LIN {X 0,Y 417.271,Z 465.296,A -85,B 0,C 180,E1 -10175.316,E2 -10175.316} C_VEL
LIN {X 0,Y 417.317,Z 461.12,A -85,B 0,C 180,E1 -10176.771,E2 -10176.771} C_VEL
LIN {X 0,Y 417.422,Z 454.683,A -85,B 0,C 180,E1 -10178.472,E2 -10178.472} C_VEL
LIN {X 0,Y 417.63,Z 447.667,A -85,B 0,C 180,E1 -10179.933,E2 -10179.933} C_VEL
LIN {X 0,Y 418.109,Z 438.94,A -85,B 0,C 180,E1 -10181.392,E2 -10181.392} C_VEL
LIN {X 0,Y 418.694,Z 429.948,A -85,B 0,C 180,E1 -10182.605,E2 -10182.605} C_VEL
LIN {X 0,Y 419.338,Z 418.893,A -85,B 0,C 180,E1 -10183.818,E2 -10183.818} C_VEL
LIN {X 0,Y 420.032,Z 407.756,A -85,B 0,C 180,E1 -10184.784,E2 -10184.784} C_VEL
LIN {X 0,Y 420.914,Z 395.292,A -85,B 0,C 180,E1 -10185.62,E2 -10185.62} C_VEL
LIN {X 0,Y 421.545,Z 382.66,A -85,B 0,C 180,E1 -10186.247,E2 -10186.247} C_VEL
LIN {X 0,Y 422.133,Z 369.345,A -85,B 0,C 180,E1 -10186.69,E2 -10186.69} C_VEL
LIN {X 0,Y 423.204,Z 286.093,A -85,B 0,C 180,E1 -10188.305,E2 -10188.305} C_VEL
LIN {X 0,Y 420.595,Z 264.034,A -85,B 0,C 180,E1 -10188.899,E2 -10188.899} C_VEL
LIN {X 0,Y 420.271,Z 261.318,A -85,B 0,C 180,E1 -10189.016,E2 -10189.016} C_VEL
LIN {X 0,Y 421.665,Z 236.885,A -85,B 0,C 180,E1 -10192.542,E2 -10192.542} C_VEL
LIN {X 0,Y 423.214,Z 213.553,A -85,B 0,C 180,E1 -10195.973,E2 -10195.973} C_VEL
LIN {X 0,Y 420.894,Z 202.341,A -85,B 0,C 180,E1 -10197.875,E2 -10197.875} C_VEL
LIN {X 0,Y 418.276,Z 192.511,A -85,B 0,C 180,E1 -10199.696,E2 -10199.696} C_VEL
LIN {X 0,Y 418.261,Z 192.387,A -85,B 0,C 180,E1 -10202.844,E2 -10202.844} C_VEL
LIN {X 0,Y 418.247,Z 192.387,A -85,B 0,C 180,E1 -10206.238,E2 -10206.238} C_VEL
LIN {X 0,Y 418.203,Z 192.393,A -85,B 0,C 180,E1 -10209.688,E2 -10209.688} C_VEL
LIN {X 0,Y 418.215,Z 192.39,A -85,B 0,C 180,E1 -10212.318,E2 -10212.318} C_VEL
LIN {X 0,Y 418.239,Z 192.391,A -85,B 0,C 180,E1 -10215.109,E2 -10215.109} C_VEL
LIN {X 0,Y 418.237,Z 192.384,A -85,B 0,C 180,E1 -10217.766,E2 -10217.766} C_VEL
LIN {X 0,Y 418.248,Z 192.385,A -85,B 0,C 180,E1 -10220.621,E2 -10220.621} C_VEL
LIN {X 0,Y 418.245,Z 192.384,A -85,B 0,C 180,E1 -10223.976,E2 -10223.976} C_VEL
LIN {X 0,Y 418.26,Z 192.386,A -85,B 0,C 180,E1 -10227.156,E2 -10227.156} C_VEL
LIN {X 0,Y 418.271,Z 192.383,A -85,B 0,C 180,E1 -10230.895,E2 -10230.895} C_VEL
LIN {X 0,Y 418.271,Z 192.383,A -85,B 0,C 180,E1 -10234.095,E2 -10234.095} C_VEL
LIN {X 0,Y 418.24,Z 192.386,A -85,B 0,C 180,E1 -10237.263,E2 -10237.263} C_VEL
LIN {X 0,Y 418.285,Z 192.385,A -85,B 0,C 180,E1 -10240.364,E2 -10240.364} C_VEL
LIN {X 0,Y 418.318,Z 192.377,A -85,B 0,C 180,E1 -10243.404,E2 -10243.404} C_VEL
LIN {X 0,Y 418.348,Z 192.373,A -85,B 0,C 180,E1 -10246.999,E2 -10246.999} C_VEL
LIN {X 0,Y 418.341,Z 192.377,A -85,B 0,C 180,E1 -10250.328,E2 -10250.328} C_VEL
LIN {X 0,Y 418.46,Z 192.36,A -85,B 0,C 180,E1 -10253.248,E2 -10253.248} C_VEL
LIN {X 0,Y 418.334,Z 192.378,A -85,B 0,C 180,E1 -10255.181,E2 -10255.181} C_VEL
LIN {X 0,Y 418.456,Z 192.55,A -85,B 0,C 180,E1 -10256.871,E2 -10256.871} C_VEL
LIN {X 0,Y 420.63,Z 201.709,A -85,B 0,C 180,E1 -10258.803,E2 -10258.803} C_VEL
LIN {X 0,Y 420.547,Z 211.888,A -85,B 0,C 180,E1 -10260.718,E2 -10260.718} C_VEL
LIN {X 0,Y 420.179,Z 229.574,A -85,B 0,C 180,E1 -10264.016,E2 -10264.016} C_VEL
LIN {X 0,Y 423.338,Z 244.848,A -85,B 0,C 180,E1 -10264.582,E2 -10264.582} C_VEL
LIN {X 0,Y 421.949,Z 313.811,A -85,B 0,C 180,E1 -10266.125,E2 -10266.125} C_VEL
LIN {X 0,Y 421.711,Z 325.601,A -85,B 0,C 180,E1 -10266.579,E2 -10266.579} C_VEL
LIN {X 0,Y 421.311,Z 336.524,A -85,B 0,C 180,E1 -10267.187,E2 -10267.187} C_VEL
LIN {X 0,Y 420.865,Z 346.473,A -85,B 0,C 180,E1 -10267.918,E2 -10267.918} C_VEL
LIN {X 0,Y 420.345,Z 356.216,A -85,B 0,C 180,E1 -10268.841,E2 -10268.841} C_VEL
LIN {X 0,Y 419.827,Z 364.922,A -85,B 0,C 180,E1 -10269.88,E2 -10269.88} C_VEL
LIN {X 0,Y 419.243,Z 373.147,A -85,B 0,C 180,E1 -10271.115,E2 -10271.115} C_VEL
LIN {X 0,Y 418.796,Z 379.629,A -85,B 0,C 180,E1 -10272.354,E2 -10272.354} C_VEL
LIN {X 0,Y 418.393,Z 384.792,A -85,B 0,C 180,E1 -10273.601,E2 -10273.601} C_VEL
LIN {X 0,Y 418.019,Z 389.504,A -85,B 0,C 180,E1 -10275.105,E2 -10275.105} C_VEL
LIN {X 0,Y 417.796,Z 392.747,A -85,B 0,C 180,E1 -10276.616,E2 -10276.616} C_VEL
LIN {X 0,Y 417.651,Z 394.16,A -85,B 0,C 180,E1 -10277.631,E2 -10277.631} C_VEL
LIN {X 0,Y 417.524,Z 395.021,A -85,B 0,C 180,E1 -10278.651,E2 -10278.651} C_VEL
LIN {X 0,Y 417.469,Z 395.273,A -85,B 0,C 180,E1 -10279.675,E2 -10279.675} C_VEL
LIN {X 0,Y 417.425,Z 394.957,A -85,B 0,C 180,E1 -10280.705,E2 -10280.705} C_VEL
LIN {X 0,Y 417.497,Z 393.456,A -85,B 0,C 180,E1 -10282.203,E2 -10282.203} C_VEL
LIN {X 0,Y 417.655,Z 390.389,A -85,B 0,C 180,E1 -10283.819,E2 -10283.819} C_VEL
LIN {X 0,Y 417.803,Z 387.549,A -85,B 0,C 180,E1 -10284.868,E2 -10284.868} C_VEL
LIN {X 0,Y 418.077,Z 381.826,A -85,B 0,C 180,E1 -10286.453,E2 -10286.453} C_VEL
LIN {X 0,Y 418.354,Z 375.584,A -85,B 0,C 180,E1 -10287.759,E2 -10287.759} C_VEL
LIN {X 0,Y 418.706,Z 369.068,A -85,B 0,C 180,E1 -10288.853,E2 -10288.853} C_VEL
LIN {X 0,Y 419.139,Z 360.148,A -85,B 0,C 180,E1 -10290.05,E2 -10290.05} C_VEL
LIN {X 0,Y 419.518,Z 351.23,A -85,B 0,C 180,E1 -10291.006,E2 -10291.006} C_VEL
LIN {X 0,Y 419.96,Z 340.418,A -85,B 0,C 180,E1 -10291.911,E2 -10291.911} C_VEL
LIN {X 0,Y 420.333,Z 328.992,A -85,B 0,C 180,E1 -10292.63,E2 -10292.63} C_VEL
LIN {X 0,Y 420.541,Z 317.102,A -85,B 0,C 180,E1 -10293.164,E2 -10293.164} C_VEL
LIN {X 0,Y 420.702,Z 305.658,A -85,B 0,C 180,E1 -10293.49,E2 -10293.49} C_VEL
LIN {X 0,Y 421.451,Z 242.868,A -85,B 0,C 180,E1 -10294.748,E2 -10294.748} C_VEL
LIN {X 0,Y 419.042,Z 228.513,A -85,B 0,C 180,E1 -10295.14,E2 -10295.14} C_VEL
LIN {X 0,Y 419.063,Z 227.046,A -85,B 0,C 180,E1 -10295.35,E2 -10295.35} C_VEL
LIN {X 0,Y 419.499,Z 211.477,A -85,B 0,C 180,E1 -10298.613,E2 -10298.613} C_VEL
LIN {X 0,Y 419.772,Z 201.372,A -85,B 0,C 180,E1 -10300.764,E2 -10300.764} C_VEL
LIN {X 0,Y 418.633,Z 194.184,A -85,B 0,C 180,E1 -10302.381,E2 -10302.381} C_VEL
LIN {X 0,Y 418.268,Z 192.411,A -85,B 0,C 180,E1 -10302.87,E2 -10302.87} C_VEL
LIN {X 0,Y 418.208,Z 192.392,A -85,B 0,C 180,E1 -10306.27,E2 -10306.27} C_VEL
LIN {X 0,Y 418.221,Z 192.387,A -85,B 0,C 180,E1 -10309.13,E2 -10309.13} C_VEL
LIN {X 0,Y 418.225,Z 192.387,A -85,B 0,C 180,E1 -10312.166,E2 -10312.166} C_VEL
LIN {X 0,Y 418.264,Z 192.385,A -85,B 0,C 180,E1 -10315.419,E2 -10315.419} C_VEL
LIN {X 0,Y 418.209,Z 192.387,A -85,B 0,C 180,E1 -10318.603,E2 -10318.603} C_VEL
LIN {X 0,Y 418.291,Z 192.379,A -85,B 0,C 180,E1 -10321.936,E2 -10321.936} C_VEL
LIN {X 0,Y 418.288,Z 192.381,A -85,B 0,C 180,E1 -10325.162,E2 -10325.162} C_VEL
LIN {X 0,Y 418.232,Z 192.384,A -85,B 0,C 180,E1 -10328.303,E2 -10328.303} C_VEL
LIN {X 0,Y 418.282,Z 192.385,A -85,B 0,C 180,E1 -10331.383,E2 -10331.383} C_VEL
LIN {X 0,Y 418.291,Z 192.377,A -85,B 0,C 180,E1 -10334.036,E2 -10334.036} C_VEL
LIN {X 0,Y 417.64,Z 192.462,A -85,B 0,C 180,E1 -10334.84,E2 -10334.84} C_VEL
LIN {X 0,Y 414.816,Z 192.81,A -85,B 0,C 180,E1 -10336.148,E2 -10336.148} C_VEL
LIN {X 0,Y 412.412,Z 193.115,A -85,B 0,C 180,E1 -10337.203,E2 -10337.203} C_VEL
LIN {X 0,Y 411.367,Z 193.24,A -85,B 0,C 180,E1 -10338.019,E2 -10338.019} C_VEL
LIN {X 0,Y 411.276,Z 193.251,A -85,B 0,C 180,E1 -10338.295,E2 -10338.295} C_VEL
LIN {X 0,Y 411.48,Z 193.225,A -85,B 0,C 180,E1 -10342.146,E2 -10342.146} C_VEL
LIN {X 0,Y 411.474,Z 193.226,A -85,B 0,C 180,E1 -10344.117,E2 -10344.117} C_VEL
LIN {X 0,Y 411.511,Z 193.221,A -85,B 0,C 180,E1 -10348.042,E2 -10348.042} C_VEL
LIN {X 0,Y 411.64,Z 193.205,A -85,B 0,C 180,E1 -10349.999,E2 -10349.999} C_VEL
LIN {X 0,Y 411.463,Z 193.233,A -85,B 0,C 180,E1 -10352.936,E2 -10352.936} C_VEL
LIN {X 0,Y 411.448,Z 193.235,A -85,B 0,C 180,E1 -10356.866,E2 -10356.866} C_VEL
LIN {X 0,Y 411.29,Z 193.249,A -85,B 0,C 180,E1 -10359.838,E2 -10359.838} C_VEL
LIN {X 0,Y 411.301,Z 193.252,A -85,B 0,C 180,E1 -10363.103,E2 -10363.103} C_VEL
LIN {X 0,Y 411.253,Z 193.26,A -85,B 0,C 180,E1 -10366.888,E2 -10366.888} C_VEL
LIN {X 0,Y 411.225,Z 193.257,A -85,B 0,C 180,E1 -10369.986,E2 -10369.986} C_VEL
LIN {X 0,Y 411.198,Z 193.263,A -85,B 0,C 180,E1 -10373.147,E2 -10373.147} C_VEL
LIN {X 0,Y 411.233,Z 193.26,A -85,B 0,C 180,E1 -10376.38,E2 -10376.38} C_VEL
LIN {X 0,Y 411.194,Z 193.261,A -85,B 0,C 180,E1 -10379.712,E2 -10379.712} C_VEL
LIN {X 0,Y 411.2,Z 193.261,A -85,B 0,C 180,E1 -10383.155,E2 -10383.155} C_VEL
LIN {X 0,Y 411.189,Z 193.268,A -85,B 0,C 180,E1 -10386.553,E2 -10386.553} C_VEL
LIN {X 0,Y 411.22,Z 193.258,A -85,B 0,C 180,E1 -10389.73,E2 -10389.73} C_VEL
LIN {X 0,Y 411.214,Z 193.259,A -85,B 0,C 180,E1 -10393.127,E2 -10393.127} C_VEL
LIN {X 0,Y 411.165,Z 193.266,A -85,B 0,C 180,E1 -10395.88,E2 -10395.88} C_VEL
LIN {X 0,Y 411.203,Z 193.26,A -85,B 0,C 180,E1 -10399.499,E2 -10399.499} C_VEL
LIN {X 0,Y 411.195,Z 193.265,A -85,B 0,C 180,E1 -10402.027,E2 -10402.027} C_VEL
LIN {X 0,Y 411.198,Z 193.262,A -85,B 0,C 180,E1 -10405.666,E2 -10405.666} C_VEL
LIN {X 0,Y 411.193,Z 193.261,A -85,B 0,C 180,E1 -10409.153,E2 -10409.153} C_VEL
LIN {X 0,Y 411.251,Z 193.256,A -85,B 0,C 180,E1 -10412.522,E2 -10412.522} C_VEL
LIN {X 0,Y 411.218,Z 193.262,A -85,B 0,C 180,E1 -10415.785,E2 -10415.785} C_VEL
LIN {X 0,Y 411.188,Z 193.262,A -85,B 0,C 180,E1 -10418.966,E2 -10418.966} C_VEL
LIN {X 0,Y 411.245,Z 193.26,A -85,B 0,C 180,E1 -10422.085,E2 -10422.085} C_VEL
LIN {X 0,Y 411.256,Z 193.253,A -85,B 0,C 180,E1 -10425.148,E2 -10425.148} C_VEL
LIN {X 0,Y 411.276,Z 193.254,A -85,B 0,C 180,E1 -10428.168,E2 -10428.168} C_VEL
LIN {X 0,Y 411.432,Z 193.234,A -85,B 0,C 180,E1 -10432.189,E2 -10432.189} C_VEL
LIN {X 0,Y 411.466,Z 193.23,A -85,B 0,C 180,E1 -10434.118,E2 -10434.118} C_VEL
LIN {X 0,Y 411.502,Z 193.226,A -85,B 0,C 180,E1 -10438.043,E2 -10438.043} C_VEL
LIN {X 0,Y 411.633,Z 193.209,A -85,B 0,C 180,E1 -10440,E2 -10440} C_VEL
LIN {X 0,Y 411.45,Z 193.23,A -85,B 0,C 180,E1 -10442.938,E2 -10442.938} C_VEL
LIN {X 0,Y 411.45,Z 193.23,A -85,B 0,C 180,E1 -10446.868,E2 -10446.868} C_VEL
LIN {X 0,Y 411.346,Z 193.243,A -85,B 0,C 180,E1 -10448.846,E2 -10448.846} C_VEL
LIN {X 0,Y 411.276,Z 193.254,A -85,B 0,C 180,E1 -10451.833,E2 -10451.833} C_VEL
LIN {X 0,Y 411.252,Z 193.255,A -85,B 0,C 180,E1 -10454.853,E2 -10454.853} C_VEL
LIN {X 0,Y 411.245,Z 193.256,A -85,B 0,C 180,E1 -10457.916,E2 -10457.916} C_VEL
LIN {X 0,Y 411.19,Z 193.265,A -85,B 0,C 180,E1 -10461.035,E2 -10461.035} C_VEL
LIN {X 0,Y 411.22,Z 193.258,A -85,B 0,C 180,E1 -10464.216,E2 -10464.216} C_VEL
LIN {X 0,Y 411.253,Z 193.258,A -85,B 0,C 180,E1 -10467.479,E2 -10467.479} C_VEL
LIN {X 0,Y 411.183,Z 193.265,A -85,B 0,C 180,E1 -10470.849,E2 -10470.849} C_VEL
LIN {X 0,Y 411.199,Z 193.26,A -85,B 0,C 180,E1 -10474.335,E2 -10474.335} C_VEL
LIN {X 0,Y 411.188,Z 193.262,A -85,B 0,C 180,E1 -10477.975,E2 -10477.975} C_VEL
LIN {X 0,Y 411.159,Z 193.27,A -85,B 0,C 180,E1 -10481.229,E2 -10481.229} C_VEL
LIN {X 0,Y 411.172,Z 193.265,A -85,B 0,C 180,E1 -10484.491,E2 -10484.491} C_VEL
LIN {X 0,Y 411.17,Z 193.264,A -85,B 0,C 180,E1 -10488.195,E2 -10488.195} C_VEL
LIN {X 0,Y 411.208,Z 193.265,A -85,B 0,C 180,E1 -10490.776,E2 -10490.776} C_VEL
LIN {X 0,Y 411.195,Z 193.264,A -85,B 0,C 180,E1 -10494.472,E2 -10494.472} C_VEL
LIN {X 0,Y 411.206,Z 193.266,A -85,B 0,C 180,E1 -10496.874,E2 -10496.874} C_VEL
LIN {X 0,Y 411.263,Z 193.447,A -85,B 0,C 180,E1 -10500.405,E2 -10500.405} C_VEL
LIN {X 0,Y 415.049,Z 210.098,A -85,B 0,C 180,E1 -10503.317,E2 -10503.317} C_VEL
LIN {X 0,Y 415.807,Z 213.749,A -85,B 0,C 180,E1 -10503.932,E2 -10503.932} C_VEL
LIN {X 0,Y 414.983,Z 228.074,A -85,B 0,C 180,E1 -10506.139,E2 -10506.139} C_VEL
LIN {X 0,Y 413.235,Z 254.249,A -85,B 0,C 180,E1 -10510.115,E2 -10510.115} C_VEL
LIN {X 0,Y 412.767,Z 263.296,A -85,B 0,C 180,E1 -10511.448,E2 -10511.448} C_VEL
LIN {X 0,Y 415.274,Z 288.029,A -85,B 0,C 180,E1 -10512.03,E2 -10512.03} C_VEL
LIN {X 0,Y 414.314,Z 370.3,A -85,B 0,C 180,E1 -10513.589,E2 -10513.589} C_VEL
LIN {X 0,Y 413.823,Z 383.827,A -85,B 0,C 180,E1 -10514.044,E2 -10514.044} C_VEL
LIN {X 0,Y 413.289,Z 396.045,A -85,B 0,C 180,E1 -10514.655,E2 -10514.655} C_VEL
LIN {X 0,Y 412.62,Z 407.808,A -85,B 0,C 180,E1 -10515.45,E2 -10515.45} C_VEL
LIN {X 0,Y 412,Z 418.559,A -85,B 0,C 180,E1 -10516.378,E2 -10516.378} C_VEL
LIN {X 0,Y 411.554,Z 428.336,A -85,B 0,C 180,E1 -10517.425,E2 -10517.425} C_VEL
LIN {X 0,Y 411.037,Z 435.948,A -85,B 0,C 180,E1 -10518.411,E2 -10518.411} C_VEL
LIN {X 0,Y 410.635,Z 443.931,A -85,B 0,C 180,E1 -10519.648,E2 -10519.648} C_VEL
LIN {X 0,Y 410.332,Z 451.666,A -85,B 0,C 180,E1 -10521.133,E2 -10521.133} C_VEL
LIN {X 0,Y 410.256,Z 457.854,A -85,B 0,C 180,E1 -10522.619,E2 -10522.619} C_VEL
LIN {X 0,Y 410.195,Z 462.697,A -85,B 0,C 180,E1 -10524.1,E2 -10524.1} C_VEL
LIN {X 0,Y 410.153,Z 466.343,A -85,B 0,C 180,E1 -10525.578,E2 -10525.578} C_VEL
LIN {X 0,Y 410.337,Z 468.924,A -85,B 0,C 180,E1 -10527.055,E2 -10527.055} C_VEL
LIN {X 0,Y 410.289,Z 470.074,A -85,B 0,C 180,E1 -10528.037,E2 -10528.037} C_VEL
LIN {X 0,Y 410.211,Z 470.747,A -85,B 0,C 180,E1 -10529.019,E2 -10529.019} C_VEL
LIN {X 0,Y 410.211,Z 471.014,A -85,B 0,C 180,E1 -10530.001,E2 -10530.001} C_VEL
LIN {X 0,Y 410.212,Z 470.867,A -85,B 0,C 180,E1 -10530.982,E2 -10530.982} C_VEL
LIN {X 0,Y 410.287,Z 470.264,A -85,B 0,C 180,E1 -10531.964,E2 -10531.964} C_VEL
LIN {X 0,Y 410.293,Z 469.224,A -85,B 0,C 180,E1 -10532.946,E2 -10532.946} C_VEL
LIN {X 0,Y 410.208,Z 467.759,A -85,B 0,C 180,E1 -10533.93,E2 -10533.93} C_VEL
LIN {X 0,Y 410.177,Z 464.691,A -85,B 0,C 180,E1 -10535.408,E2 -10535.408} C_VEL
LIN {X 0,Y 410.25,Z 460.536,A -85,B 0,C 180,E1 -10536.888,E2 -10536.888} C_VEL
LIN {X 0,Y 410.332,Z 454.126,A -85,B 0,C 180,E1 -10538.62,E2 -10538.62} C_VEL
LIN {X 0,Y 410.577,Z 447.128,A -85,B 0,C 180,E1 -10540.106,E2 -10540.106} C_VEL
LIN {X 0,Y 411.103,Z 438.459,A -85,B 0,C 180,E1 -10541.589,E2 -10541.589} C_VEL
LIN {X 0,Y 411.731,Z 429.519,A -85,B 0,C 180,E1 -10542.821,E2 -10542.821} C_VEL
LIN {X 0,Y 412.344,Z 419.718,A -85,B 0,C 180,E1 -10543.931,E2 -10543.931} C_VEL
LIN {X 0,Y 413.035,Z 409.012,A -85,B 0,C 180,E1 -10544.914,E2 -10544.914} C_VEL
LIN {X 0,Y 413.956,Z 397.074,A -85,B 0,C 180,E1 -10545.763,E2 -10545.763} C_VEL
LIN {X 0,Y 414.627,Z 384.67,A -85,B 0,C 180,E1 -10546.431,E2 -10546.431} C_VEL
LIN {X 0,Y 415.25,Z 371.848,A -85,B 0,C 180,E1 -10546.912,E2 -10546.912} C_VEL
LIN {X 0,Y 415.607,Z 355.316,A -85,B 0,C 180,E1 -10547.277,E2 -10547.277} C_VEL
LIN {X 0,Y 416.552,Z 286.903,A -85,B 0,C 180,E1 -10548.625,E2 -10548.625} C_VEL
LIN {X 0,Y 413.948,Z 264.743,A -85,B 0,C 180,E1 -10549.243,E2 -10549.243} C_VEL
LIN {X 0,Y 413.453,Z 261.191,A -85,B 0,C 180,E1 -10549.365,E2 -10549.365} C_VEL
LIN {X 0,Y 414.945,Z 236.899,A -85,B 0,C 180,E1 -10552.927,E2 -10552.927} C_VEL
LIN {X 0,Y 416.441,Z 216.174,A -85,B 0,C 180,E1 -10556.027,E2 -10556.027} C_VEL
LIN {X 0,Y 415.347,Z 209.331,A -85,B 0,C 180,E1 -10557.185,E2 -10557.185} C_VEL
LIN {X 0,Y 412.503,Z 197.933,A -85,B 0,C 180,E1 -10559.246,E2 -10559.246} C_VEL
LIN {X 0,Y 411.23,Z 193.377,A -85,B 0,C 180,E1 -10560.17,E2 -10560.17} C_VEL
LIN {X 0,Y 411.21,Z 193.266,A -85,B 0,C 180,E1 -10563.156,E2 -10563.156} C_VEL
LIN {X 0,Y 411.195,Z 193.267,A -85,B 0,C 180,E1 -10566.552,E2 -10566.552} C_VEL
LIN {X 0,Y 411.173,Z 193.268,A -85,B 0,C 180,E1 -10569.72,E2 -10569.72} C_VEL
LIN {X 0,Y 411.168,Z 193.27,A -85,B 0,C 180,E1 -10573.135,E2 -10573.135} C_VEL
LIN {X 0,Y 411.17,Z 193.265,A -85,B 0,C 180,E1 -10575.881,E2 -10575.881} C_VEL
LIN {X 0,Y 411.163,Z 193.269,A -85,B 0,C 180,E1 -10578.772,E2 -10578.772} C_VEL
LIN {X 0,Y 411.195,Z 193.262,A -85,B 0,C 180,E1 -10582.026,E2 -10582.026} C_VEL
LIN {X 0,Y 411.207,Z 193.261,A -85,B 0,C 180,E1 -10585.666,E2 -10585.666} C_VEL
LIN {X 0,Y 411.192,Z 193.266,A -85,B 0,C 180,E1 -10589.152,E2 -10589.152} C_VEL
LIN {X 0,Y 411.262,Z 193.257,A -85,B 0,C 180,E1 -10592.522,E2 -10592.522} C_VEL
LIN {X 0,Y 411.228,Z 193.259,A -85,B 0,C 180,E1 -10595.784,E2 -10595.784} C_VEL
LIN {X 0,Y 411.199,Z 193.263,A -85,B 0,C 180,E1 -10598.966,E2 -10598.966} C_VEL
LIN {X 0,Y 411.252,Z 193.259,A -85,B 0,C 180,E1 -10602.084,E2 -10602.084} C_VEL
LIN {X 0,Y 411.261,Z 193.257,A -85,B 0,C 180,E1 -10605.147,E2 -10605.147} C_VEL
LIN {X 0,Y 411.285,Z 193.256,A -85,B 0,C 180,E1 -10608.167,E2 -10608.167} C_VEL
LIN {X 0,Y 411.32,Z 193.249,A -85,B 0,C 180,E1 -10611.154,E2 -10611.154} C_VEL
LIN {X 0,Y 411.443,Z 193.236,A -85,B 0,C 180,E1 -10614.117,E2 -10614.117} C_VEL
LIN {X 0,Y 411.349,Z 193.482,A -85,B 0,C 180,E1 -10616.449,E2 -10616.449} C_VEL
LIN {X 0,Y 413.303,Z 200.825,A -85,B 0,C 180,E1 -10618.051,E2 -10618.051} C_VEL
LIN {X 0,Y 414.02,Z 205.585,A -85,B 0,C 180,E1 -10619.027,E2 -10619.027} C_VEL
LIN {X 0,Y 413.465,Z 223.513,A -85,B 0,C 180,E1 -10622.435,E2 -10622.435} C_VEL
LIN {X 0,Y 413.436,Z 229.89,A -85,B 0,C 180,E1 -10623.624,E2 -10623.624} C_VEL
LIN {X 0,Y 415.693,Z 240.426,A -85,B 0,C 180,E1 -10624.054,E2 -10624.054} C_VEL
LIN {X 0,Y 416.748,Z 246.964,A -85,B 0,C 180,E1 -10624.272,E2 -10624.272} C_VEL
LIN {X 0,Y 415.215,Z 314.416,A -85,B 0,C 180,E1 -10625.828,E2 -10625.828} C_VEL
LIN {X 0,Y 415.009,Z 325.435,A -85,B 0,C 180,E1 -10626.258,E2 -10626.258} C_VEL
LIN {X 0,Y 414.52,Z 337.543,A -85,B 0,C 180,E1 -10626.938,E2 -10626.938} C_VEL
LIN {X 0,Y 414.04,Z 347.396,A -85,B 0,C 180,E1 -10627.681,E2 -10627.681} C_VEL
LIN {X 0,Y 413.476,Z 357.623,A -85,B 0,C 180,E1 -10628.676,E2 -10628.676} C_VEL
LIN {X 0,Y 412.873,Z 366.66,A -85,B 0,C 180,E1 -10629.8,E2 -10629.8} C_VEL
LIN {X 0,Y 412.291,Z 374.656,A -85,B 0,C 180,E1 -10631.056,E2 -10631.056} C_VEL
LIN {X 0,Y 411.815,Z 380.982,A -85,B 0,C 180,E1 -10632.317,E2 -10632.317} C_VEL
LIN {X 0,Y 411.308,Z 386.876,A -85,B 0,C 180,E1 -10633.84,E2 -10633.84} C_VEL
LIN {X 0,Y 410.947,Z 391.186,A -85,B 0,C 180,E1 -10635.371,E2 -10635.371} C_VEL
LIN {X 0,Y 410.689,Z 394.048,A -85,B 0,C 180,E1 -10636.912,E2 -10636.912} C_VEL
LIN {X 0,Y 410.552,Z 395.252,A -85,B 0,C 180,E1 -10637.946,E2 -10637.946} C_VEL
LIN {X 0,Y 410.416,Z 395.943,A -85,B 0,C 180,E1 -10639.639,E2 -10639.639} C_VEL
LIN {X 0,Y 410.375,Z 395.356,A -85,B 0,C 180,E1 -10641.078,E2 -10641.078} C_VEL
LIN {X 0,Y 410.43,Z 393.848,A -85,B 0,C 180,E1 -10642.381,E2 -10642.381} C_VEL
LIN {X 0,Y 410.59,Z 391.312,A -85,B 0,C 180,E1 -10643.718,E2 -10643.718} C_VEL
LIN {X 0,Y 410.819,Z 386.889,A -85,B 0,C 180,E1 -10645.32,E2 -10645.32} C_VEL
LIN {X 0,Y 411.078,Z 381.079,A -85,B 0,C 180,E1 -10646.833,E2 -10646.833} C_VEL
LIN {X 0,Y 411.36,Z 375.246,A -85,B 0,C 180,E1 -10648.023,E2 -10648.023} C_VEL
LIN {X 0,Y 411.775,Z 367.279,A -85,B 0,C 180,E1 -10649.31,E2 -10649.31} C_VEL
LIN {X 0,Y 412.251,Z 358.167,A -85,B 0,C 180,E1 -10650.475,E2 -10650.475} C_VEL
LIN {X 0,Y 412.678,Z 348.902,A -85,B 0,C 180,E1 -10651.416,E2 -10651.416} C_VEL
LIN {X 0,Y 413.11,Z 338.264,A -85,B 0,C 180,E1 -10652.26,E2 -10652.26} C_VEL
LIN {X 0,Y 413.462,Z 326.648,A -85,B 0,C 180,E1 -10652.951,E2 -10652.951} C_VEL
LIN {X 0,Y 413.66,Z 314.08,A -85,B 0,C 180,E1 -10653.468,E2 -10653.468} C_VEL
LIN {X 0,Y 413.903,Z 296.181,A -85,B 0,C 180,E1 -10653.879,E2 -10653.879} C_VEL
LIN {X 0,Y 414.572,Z 243.794,A -85,B 0,C 180,E1 -10654.959,E2 -10654.959} C_VEL
LIN {X 0,Y 412.07,Z 228.591,A -85,B 0,C 180,E1 -10655.381,E2 -10655.381} C_VEL
LIN {X 0,Y 412.294,Z 220.823,A -85,B 0,C 180,E1 -10656.951,E2 -10656.951} C_VEL
LIN {X 0,Y 412.804,Z 203.589,A -85,B 0,C 180,E1 -10660.632,E2 -10660.632} C_VEL
LIN {X 0,Y 412.137,Z 197.789,A -85,B 0,C 180,E1 -10661.934,E2 -10661.934} C_VEL
LIN {X 0,Y 411.244,Z 193.317,A -85,B 0,C 180,E1 -10663.033,E2 -10663.033} C_VEL
LIN {X 0,Y 411.172,Z 193.267,A -85,B 0,C 180,E1 -10666.866,E2 -10666.866} C_VEL
LIN {X 0,Y 411.208,Z 193.26,A -85,B 0,C 180,E1 -10670.272,E2 -10670.272} C_VEL
LIN {X 0,Y 411.191,Z 193.266,A -85,B 0,C 180,E1 -10673.447,E2 -10673.447} C_VEL
LIN {X 0,Y 411.206,Z 193.26,A -85,B 0,C 180,E1 -10676.873,E2 -10676.873} C_VEL
LIN {X 0,Y 411.231,Z 193.256,A -85,B 0,C 180,E1 -10680.644,E2 -10680.644} C_VEL
LIN {X 0,Y 411.237,Z 193.261,A -85,B 0,C 180,E1 -10683.619,E2 -10683.619} C_VEL
LIN {X 0,Y 411.202,Z 193.261,A -85,B 0,C 180,E1 -10686.852,E2 -10686.852} C_VEL
LIN {X 0,Y 411.213,Z 193.259,A -85,B 0,C 180,E1 -10690.05,E2 -10690.05} C_VEL
LIN {X 0,Y 411.261,Z 193.257,A -85,B 0,C 180,E1 -10693.131,E2 -10693.131} C_VEL
LIN {X 0,Y 411.304,Z 193.25,A -85,B 0,C 180,E1 -10696.895,E2 -10696.895} C_VEL
LIN {X 0,Y 411.276,Z 193.251,A -85,B 0,C 180,E1 -10698.295,E2 -10698.295} C_VEL
LIN {X 0,Y 410.61,Z 193.339,A -85,B 0,C 180,E1 -10699.112,E2 -10699.112} C_VEL
LIN {X 0,Y 407.832,Z 193.68,A -85,B 0,C 180,E1 -10700.443,E2 -10700.443} C_VEL
LIN {X 0,Y 405.492,Z 193.975,A -85,B 0,C 180,E1 -10701.518,E2 -10701.518} C_VEL
LIN {X 0,Y 404.488,Z 194.097,A -85,B 0,C 180,E1 -10702.347,E2 -10702.347} C_VEL
LIN {X 0,Y 404.406,Z 194.108,A -85,B 0,C 180,E1 -10702.628,E2 -10702.628} C_VEL
LIN {X 0,Y 404.281,Z 194.127,A -85,B 0,C 180,E1 -10705.013,E2 -10705.013} C_VEL
LIN {X 0,Y 404.48,Z 194.097,A -85,B 0,C 180,E1 -10708.008,E2 -10708.008} C_VEL
LIN {X 0,Y 404.609,Z 194.081,A -85,B 0,C 180,E1 -10709.999,E2 -10709.999} C_VEL
LIN {X 0,Y 404.42,Z 194.111,A -85,B 0,C 180,E1 -10712.988,E2 -10712.988} C_VEL
LIN {X 0,Y 404.396,Z 194.115,A -85,B 0,C 180,E1 -10716.987,E2 -10716.987} C_VEL
LIN {X 0,Y 404.255,Z 194.125,A -85,B 0,C 180,E1 -10720.011,E2 -10720.011} C_VEL
LIN {X 0,Y 404.262,Z 194.128,A -85,B 0,C 180,E1 -10723.211,E2 -10723.211} C_VEL
LIN {X 0,Y 404.211,Z 194.136,A -85,B 0,C 180,E1 -10727.006,E2 -10727.006} C_VEL
LIN {X 0,Y 404.159,Z 194.14,A -85,B 0,C 180,E1 -10730.351,E2 -10730.351} C_VEL
LIN {X 0,Y 404.164,Z 194.137,A -85,B 0,C 180,E1 -10733.574,E2 -10733.574} C_VEL
LIN {X 0,Y 404.178,Z 194.135,A -85,B 0,C 180,E1 -10735.766,E2 -10735.766} C_VEL
LIN {X 0,Y 404.19,Z 194.134,A -85,B 0,C 180,E1 -10737.999,E2 -10737.999} C_VEL
LIN {X 0,Y 404.133,Z 194.14,A -85,B 0,C 180,E1 -10741.557,E2 -10741.557} C_VEL
LIN {X 0,Y 404.181,Z 194.136,A -85,B 0,C 180,E1 -10745.015,E2 -10745.015} C_VEL
LIN {X 0,Y 404.156,Z 194.141,A -85,B 0,C 180,E1 -10748.755,E2 -10748.755} C_VEL
LIN {X 0,Y 404.184,Z 194.134,A -85,B 0,C 180,E1 -10751.61,E2 -10751.61} C_VEL
LIN {X 0,Y 404.181,Z 194.14,A -85,B 0,C 180,E1 -10754.528,E2 -10754.528} C_VEL
LIN {X 0,Y 404.164,Z 194.137,A -85,B 0,C 180,E1 -10757.3,E2 -10757.3} C_VEL
LIN {X 0,Y 404.16,Z 194.14,A -85,B 0,C 180,E1 -10759.955,E2 -10759.955} C_VEL
LIN {X 0,Y 404.132,Z 194.141,A -85,B 0,C 180,E1 -10763.124,E2 -10763.124} C_VEL
LIN {X 0,Y 404.137,Z 194.147,A -85,B 0,C 180,E1 -10766.188,E2 -10766.188} C_VEL
LIN {X 0,Y 404.156,Z 194.14,A -85,B 0,C 180,E1 -10769.716,E2 -10769.716} C_VEL
LIN {X 0,Y 404.187,Z 194.134,A -85,B 0,C 180,E1 -10773.123,E2 -10773.123} C_VEL
LIN {X 0,Y 404.168,Z 194.137,A -85,B 0,C 180,E1 -10775.334,E2 -10775.334} C_VEL
LIN {X 0,Y 404.13,Z 194.142,A -85,B 0,C 180,E1 -10778.581,E2 -10778.581} C_VEL
LIN {X 0,Y 404.202,Z 194.137,A -85,B 0,C 180,E1 -10781.762,E2 -10781.762} C_VEL
LIN {X 0,Y 404.203,Z 194.132,A -85,B 0,C 180,E1 -10784.882,E2 -10784.882} C_VEL
LIN {X 0,Y 404.248,Z 194.132,A -85,B 0,C 180,E1 -10787.959,E2 -10787.959} C_VEL
LIN {X 0,Y 404.396,Z 194.111,A -85,B 0,C 180,E1 -10792.129,E2 -10792.129} C_VEL
LIN {X 0,Y 404.414,Z 194.11,A -85,B 0,C 180,E1 -10794.015,E2 -10794.015} C_VEL
LIN {X 0,Y 404.471,Z 194.102,A -85,B 0,C 180,E1 -10798.009,E2 -10798.009} C_VEL
LIN {X 0,Y 404.603,Z 194.085,A -85,B 0,C 180,E1 -10800,E2 -10800} C_VEL
LIN {X 0,Y 404.408,Z 194.107,A -85,B 0,C 180,E1 -10802.989,E2 -10802.989} C_VEL
LIN {X 0,Y 404.402,Z 194.108,A -85,B 0,C 180,E1 -10806.988,E2 -10806.988} C_VEL
LIN {X 0,Y 404.25,Z 194.128,A -85,B 0,C 180,E1 -10810.012,E2 -10810.012} C_VEL
LIN {X 0,Y 404.259,Z 194.129,A -85,B 0,C 180,E1 -10813.212,E2 -10813.212} C_VEL
LIN {X 0,Y 404.209,Z 194.134,A -85,B 0,C 180,E1 -10817.008,E2 -10817.008} C_VEL
LIN {X 0,Y 404.157,Z 194.137,A -85,B 0,C 180,E1 -10820.352,E2 -10820.352} C_VEL
LIN {X 0,Y 404.163,Z 194.141,A -85,B 0,C 180,E1 -10823.575,E2 -10823.575} C_VEL
LIN {X 0,Y 404.178,Z 194.137,A -85,B 0,C 180,E1 -10825.767,E2 -10825.767} C_VEL
LIN {X 0,Y 404.189,Z 194.134,A -85,B 0,C 180,E1 -10828.001,E2 -10828.001} C_VEL
LIN {X 0,Y 404.133,Z 194.143,A -85,B 0,C 180,E1 -10831.559,E2 -10831.559} C_VEL
LIN {X 0,Y 404.178,Z 194.141,A -85,B 0,C 180,E1 -10835.017,E2 -10835.017} C_VEL
LIN {X 0,Y 404.148,Z 194.142,A -85,B 0,C 180,E1 -10838.758,E2 -10838.758} C_VEL
LIN {X 0,Y 404.119,Z 194.144,A -85,B 0,C 180,E1 -10841.601,E2 -10841.601} C_VEL
LIN {X 0,Y 404.142,Z 194.141,A -85,B 0,C 180,E1 -10844.523,E2 -10844.523} C_VEL
LIN {X 0,Y 404.129,Z 194.144,A -85,B 0,C 180,E1 -10847.296,E2 -10847.296} C_VEL
LIN {X 0,Y 404.166,Z 194.136,A -85,B 0,C 180,E1 -10849.956,E2 -10849.956} C_VEL
LIN {X 0,Y 404.133,Z 194.147,A -85,B 0,C 180,E1 -10853.126,E2 -10853.126} C_VEL
LIN {X 0,Y 404.143,Z 194.144,A -85,B 0,C 180,E1 -10856.189,E2 -10856.189} C_VEL
LIN {X 0,Y 404.184,Z 194.184,A -85,B 0,C 180,E1 -10860.002,E2 -10860.002} C_VEL
LIN {X 0,Y 404.217,Z 194.421,A -85,B 0,C 180,E1 -10860.146,E2 -10860.146} C_VEL
LIN {X 0,Y 408.033,Z 211.112,A -85,B 0,C 180,E1 -10863.12,E2 -10863.12} C_VEL
LIN {X 0,Y 408.925,Z 216.352,A -85,B 0,C 180,E1 -10864.008,E2 -10864.008} C_VEL
LIN {X 0,Y 407.572,Z 234.948,A -85,B 0,C 180,E1 -10866.904,E2 -10866.904} C_VEL
LIN {X 0,Y 406.031,Z 258.502,A -85,B 0,C 180,E1 -10870.538,E2 -10870.538} C_VEL
LIN {X 0,Y 405.798,Z 263.033,A -85,B 0,C 180,E1 -10871.2,E2 -10871.2} C_VEL
LIN {X 0,Y 408.366,Z 288.269,A -85,B 0,C 180,E1 -10871.808,E2 -10871.808} C_VEL
LIN {X 0,Y 407.364,Z 370.139,A -85,B 0,C 180,E1 -10873.398,E2 -10873.398} C_VEL
LIN {X 0,Y 406.867,Z 383.537,A -85,B 0,C 180,E1 -10873.86,E2 -10873.86} C_VEL
LIN {X 0,Y 406.327,Z 395.164,A -85,B 0,C 180,E1 -10874.45,E2 -10874.45} C_VEL
LIN {X 0,Y 405.596,Z 407.798,A -85,B 0,C 180,E1 -10875.321,E2 -10875.321} C_VEL
LIN {X 0,Y 404.935,Z 418.877,A -85,B 0,C 180,E1 -10876.305,E2 -10876.305} C_VEL
LIN {X 0,Y 404.402,Z 429.122,A -85,B 0,C 180,E1 -10877.454,E2 -10877.454} C_VEL
LIN {X 0,Y 403.845,Z 438.215,A -85,B 0,C 180,E1 -10878.711,E2 -10878.711} C_VEL
LIN {X 0,Y 403.425,Z 445.684,A -85,B 0,C 180,E1 -10879.968,E2 -10879.968} C_VEL
LIN {X 0,Y 403.256,Z 453.001,A -85,B 0,C 180,E1 -10881.482,E2 -10881.482} C_VEL
LIN {X 0,Y 403.177,Z 458.763,A -85,B 0,C 180,E1 -10882.992,E2 -10882.992} C_VEL
LIN {X 0,Y 403.145,Z 463.238,A -85,B 0,C 180,E1 -10884.499,E2 -10884.499} C_VEL
LIN {X 0,Y 403.154,Z 466.557,A -85,B 0,C 180,E1 -10886.002,E2 -10886.002} C_VEL
LIN {X 0,Y 403.26,Z 468.187,A -85,B 0,C 180,E1 -10887.004,E2 -10887.004} C_VEL
LIN {X 0,Y 403.238,Z 469.368,A -85,B 0,C 180,E1 -10888.003,E2 -10888.003} C_VEL
LIN {X 0,Y 403.155,Z 470.062,A -85,B 0,C 180,E1 -10889.002,E2 -10889.002} C_VEL
LIN {X 0,Y 403.151,Z 470.342,A -85,B 0,C 180,E1 -10890.001,E2 -10890.001} C_VEL
LIN {X 0,Y 403.156,Z 470.209,A -85,B 0,C 180,E1 -10891,E2 -10891} C_VEL
LIN {X 0,Y 403.235,Z 469.632,A -85,B 0,C 180,E1 -10891.998,E2 -10891.998} C_VEL
LIN {X 0,Y 403.218,Z 468.601,A -85,B 0,C 180,E1 -10892.998,E2 -10892.998} C_VEL
LIN {X 0,Y 403.114,Z 467.142,A -85,B 0,C 180,E1 -10894,E2 -10894} C_VEL
LIN {X 0,Y 403.089,Z 464.093,A -85,B 0,C 180,E1 -10895.503,E2 -10895.503} C_VEL
LIN {X 0,Y 403.182,Z 459.966,A -85,B 0,C 180,E1 -10897.009,E2 -10897.009} C_VEL
LIN {X 0,Y 403.257,Z 453.601,A -85,B 0,C 180,E1 -10898.772,E2 -10898.772} C_VEL
LIN {X 0,Y 403.522,Z 446.642,A -85,B 0,C 180,E1 -10900.284,E2 -10900.284} C_VEL
LIN {X 0,Y 404.105,Z 438.012,A -85,B 0,C 180,E1 -10901.792,E2 -10901.792} C_VEL
LIN {X 0,Y 404.76,Z 429.109,A -85,B 0,C 180,E1 -10903.046,E2 -10903.046} C_VEL
LIN {X 0,Y 405.459,Z 418.145,A -85,B 0,C 180,E1 -10904.301,E2 -10904.301} C_VEL
LIN {X 0,Y 406.311,Z 407.179,A -85,B 0,C 180,E1 -10905.295,E2 -10905.295} C_VEL
LIN {X 0,Y 407.207,Z 394.874,A -85,B 0,C 180,E1 -10906.159,E2 -10906.159} C_VEL
LIN {X 0,Y 407.9,Z 383.362,A -85,B 0,C 180,E1 -10906.775,E2 -10906.775} C_VEL
LIN {X 0,Y 408.561,Z 370.177,A -85,B 0,C 180,E1 -10907.262,E2 -10907.262} C_VEL
LIN {X 0,Y 408.95,Z 348.659,A -85,B 0,C 180,E1 -10907.729,E2 -10907.729} C_VEL
LIN {X 0,Y 409.919,Z 287.437,A -85,B 0,C 180,E1 -10908.967,E2 -10908.967} C_VEL
LIN {X 0,Y 407.278,Z 265.154,A -85,B 0,C 180,E1 -10909.608,E2 -10909.608} C_VEL
LIN {X 0,Y 406.657,Z 260.583,A -85,B 0,C 180,E1 -10909.787,E2 -10909.787} C_VEL
LIN {X 0,Y 408.328,Z 235.494,A -85,B 0,C 180,E1 -10913.551,E2 -10913.551} C_VEL
LIN {X 0,Y 409.721,Z 218.043,A -85,B 0,C 180,E1 -10916.212,E2 -10916.212} C_VEL
LIN {X 0,Y 408.972,Z 212.909,A -85,B 0,C 180,E1 -10917.095,E2 -10917.095} C_VEL
LIN {X 0,Y 405.983,Z 200.542,A -85,B 0,C 180,E1 -10919.377,E2 -10919.377} C_VEL
LIN {X 0,Y 404.181,Z 194.255,A -85,B 0,C 180,E1 -10920.662,E2 -10920.662} C_VEL
LIN {X 0,Y 404.148,Z 194.145,A -85,B 0,C 180,E1 -10923.812,E2 -10923.812} C_VEL
LIN {X 0,Y 404.138,Z 194.145,A -85,B 0,C 180,E1 -10926.874,E2 -10926.874} C_VEL
LIN {X 0,Y 404.12,Z 194.146,A -85,B 0,C 180,E1 -10930.075,E2 -10930.075} C_VEL
LIN {X 0,Y 404.147,Z 194.144,A -85,B 0,C 180,E1 -10933.082,E2 -10933.082} C_VEL
LIN {X 0,Y 404.15,Z 194.14,A -85,B 0,C 180,E1 -10935.926,E2 -10935.926} C_VEL
LIN {X 0,Y 404.118,Z 194.145,A -85,B 0,C 180,E1 -10938.634,E2 -10938.634} C_VEL
LIN {X 0,Y 404.153,Z 194.14,A -85,B 0,C 180,E1 -10941.493,E2 -10941.493} C_VEL
LIN {X 0,Y 404.186,Z 194.139,A -85,B 0,C 180,E1 -10944.984,E2 -10944.984} C_VEL
LIN {X 0,Y 404.144,Z 194.141,A -85,B 0,C 180,E1 -10948.554,E2 -10948.554} C_VEL
LIN {X 0,Y 404.198,Z 194.136,A -85,B 0,C 180,E1 -10952,E2 -10952} C_VEL
LIN {X 0,Y 404.179,Z 194.137,A -85,B 0,C 180,E1 -10955.334,E2 -10955.334} C_VEL
LIN {X 0,Y 404.141,Z 194.144,A -85,B 0,C 180,E1 -10958.58,E2 -10958.58} C_VEL
LIN {X 0,Y 404.21,Z 194.134,A -85,B 0,C 180,E1 -10961.761,E2 -10961.761} C_VEL
LIN {X 0,Y 404.207,Z 194.137,A -85,B 0,C 180,E1 -10964.882,E2 -10964.882} C_VEL
LIN {X 0,Y 404.258,Z 194.129,A -85,B 0,C 180,E1 -10967.958,E2 -10967.958} C_VEL
LIN {X 0,Y 404.268,Z 194.128,A -85,B 0,C 180,E1 -10970.998,E2 -10970.998} C_VEL
LIN {X 0,Y 404.393,Z 194.114,A -85,B 0,C 180,E1 -10974.014,E2 -10974.014} C_VEL
LIN {X 0,Y 404.239,Z 194.283,A -85,B 0,C 180,E1 -10975.949,E2 -10975.949} C_VEL
LIN {X 0,Y 406.463,Z 202.326,A -85,B 0,C 180,E1 -10977.77,E2 -10977.77} C_VEL
LIN {X 0,Y 407.297,Z 207.027,A -85,B 0,C 180,E1 -10978.764,E2 -10978.764} C_VEL
LIN {X 0,Y 406.706,Z 224.999,A -85,B 0,C 180,E1 -10982.228,E2 -10982.228} C_VEL
LIN {X 0,Y 406.609,Z 230.293,A -85,B 0,C 180,E1 -10983.22,E2 -10983.22} C_VEL
LIN {X 0,Y 407.794,Z 235.677,A -85,B 0,C 180,E1 -10983.472,E2 -10983.472} C_VEL
LIN {X 0,Y 410.107,Z 246.958,A -85,B 0,C 180,E1 -10983.896,E2 -10983.896} C_VEL
LIN {X 0,Y 408.559,Z 314.42,A -85,B 0,C 180,E1 -10985.49,E2 -10985.49} C_VEL
LIN {X 0,Y 408.309,Z 325.605,A -85,B 0,C 180,E1 -10985.927,E2 -10985.927} C_VEL
LIN {X 0,Y 407.855,Z 336.819,A -85,B 0,C 180,E1 -10986.555,E2 -10986.555} C_VEL
LIN {X 0,Y 407.365,Z 346.937,A -85,B 0,C 180,E1 -10987.309,E2 -10987.309} C_VEL
LIN {X 0,Y 406.708,Z 357.374,A -85,B 0,C 180,E1 -10988.321,E2 -10988.321} C_VEL
LIN {X 0,Y 406.09,Z 366.39,A -85,B 0,C 180,E1 -10989.435,E2 -10989.435} C_VEL
LIN {X 0,Y 405.438,Z 374.759,A -85,B 0,C 180,E1 -10990.739,E2 -10990.739} C_VEL
LIN {X 0,Y 404.817,Z 382.343,A -85,B 0,C 180,E1 -10992.278,E2 -10992.278} C_VEL
LIN {X 0,Y 404.369,Z 387.372,A -85,B 0,C 180,E1 -10993.616,E2 -10993.616} C_VEL
LIN {X 0,Y 403.964,Z 391.618,A -85,B 0,C 180,E1 -10995.127,E2 -10995.127} C_VEL
LIN {X 0,Y 403.671,Z 394.668,A -85,B 0,C 180,E1 -10996.752,E2 -10996.752} C_VEL
LIN {X 0,Y 403.463,Z 396.236,A -85,B 0,C 180,E1 -10998.272,E2 -10998.272} C_VEL
LIN {X 0,Y 403.345,Z 396.612,A -85,B 0,C 180,E1 -10999.794,E2 -10999.794} C_VEL
LIN {X 0,Y 403.309,Z 395.625,A -85,B 0,C 180,E1 -11001.465,E2 -11001.465} C_VEL
LIN {X 0,Y 403.382,Z 394.177,A -85,B 0,C 180,E1 -11002.571,E2 -11002.571} C_VEL
LIN {X 0,Y 403.58,Z 390.964,A -85,B 0,C 180,E1 -11004.156,E2 -11004.156} C_VEL
LIN {X 0,Y 403.837,Z 386.057,A -85,B 0,C 180,E1 -11005.79,E2 -11005.79} C_VEL
LIN {X 0,Y 404.09,Z 380.362,A -85,B 0,C 180,E1 -11007.203,E2 -11007.203} C_VEL
LIN {X 0,Y 404.454,Z 373.419,A -85,B 0,C 180,E1 -11008.545,E2 -11008.545} C_VEL
LIN {X 0,Y 404.869,Z 365.344,A -85,B 0,C 180,E1 -11009.78,E2 -11009.78} C_VEL
LIN {X 0,Y 405.375,Z 356.119,A -85,B 0,C 180,E1 -11010.904,E2 -11010.904} C_VEL
LIN {X 0,Y 405.873,Z 345.027,A -85,B 0,C 180,E1 -11011.954,E2 -11011.954} C_VEL
LIN {X 0,Y 406.279,Z 333.194,A -85,B 0,C 180,E1 -11012.796,E2 -11012.796} C_VEL
LIN {X 0,Y 406.643,Z 321.139,A -85,B 0,C 180,E1 -11013.409,E2 -11013.409} C_VEL
LIN {X 0,Y 406.81,Z 309.466,A -85,B 0,C 180,E1 -11013.804,E2 -11013.804} C_VEL
LIN {X 0,Y 407.651,Z 244.13,A -85,B 0,C 180,E1 -11015.185,E2 -11015.185} C_VEL
LIN {X 0,Y 405.121,Z 228.936,A -85,B 0,C 180,E1 -11015.615,E2 -11015.615} C_VEL
LIN {X 0,Y 405.159,Z 226.087,A -85,B 0,C 180,E1 -11016.14,E2 -11016.14} C_VEL
LIN {X 0,Y 405.601,Z 211.542,A -85,B 0,C 180,E1 -11019.256,E2 -11019.256} C_VEL
LIN {X 0,Y 405.77,Z 202.822,A -85,B 0,C 180,E1 -11021.159,E2 -11021.159} C_VEL
LIN {X 0,Y 404.18,Z 194.215,A -85,B 0,C 180,E1 -11023.215,E2 -11023.215} C_VEL
LIN {X 0,Y 404.151,Z 194.142,A -85,B 0,C 180,E1 -11026.916,E2 -11026.916} C_VEL
LIN {X 0,Y 404.168,Z 194.14,A -85,B 0,C 180,E1 -11029.955,E2 -11029.955} C_VEL
LIN {X 0,Y 404.135,Z 194.142,A -85,B 0,C 180,E1 -11033.125,E2 -11033.125} C_VEL
LIN {X 0,Y 404.144,Z 194.14,A -85,B 0,C 180,E1 -11036.187,E2 -11036.187} C_VEL
LIN {X 0,Y 404.144,Z 194.144,A -85,B 0,C 180,E1 -11039.714,E2 -11039.714} C_VEL
LIN {X 0,Y 404.194,Z 194.136,A -85,B 0,C 180,E1 -11043.122,E2 -11043.122} C_VEL
LIN {X 0,Y 404.176,Z 194.141,A -85,B 0,C 180,E1 -11045.334,E2 -11045.334} C_VEL
LIN {X 0,Y 404.137,Z 194.14,A -85,B 0,C 180,E1 -11048.58,E2 -11048.58} C_VEL
LIN {X 0,Y 404.208,Z 194.134,A -85,B 0,C 180,E1 -11051.761,E2 -11051.761} C_VEL
LIN {X 0,Y 404.205,Z 194.134,A -85,B 0,C 180,E1 -11054.881,E2 -11054.881} C_VEL
LIN {X 0,Y 404.255,Z 194.126,A -85,B 0,C 180,E1 -11057.958,E2 -11057.958} C_VEL
LIN {X 0,Y 404.431,Z 194.103,A -85,B 0,C 180,E1 -11062.099,E2 -11062.099} C_VEL
LIN {X 0,Y 404.406,Z 194.108,A -85,B 0,C 180,E1 -11062.628,E2 -11062.628} C_VEL
LIN {X 0,Y 403.737,Z 194.198,A -85,B 0,C 180,E1 -11063.457,E2 -11063.457} C_VEL
LIN {X 0,Y 400.883,Z 194.559,A -85,B 0,C 180,E1 -11064.805,E2 -11064.805} C_VEL
LIN {X 0,Y 398.477,Z 194.858,A -85,B 0,C 180,E1 -11065.894,E2 -11065.894} C_VEL
LIN {X 0,Y 397.456,Z 194.979,A -85,B 0,C 180,E1 -11066.736,E2 -11066.736} C_VEL
LIN {X 0,Y 397.379,Z 194.986,A -85,B 0,C 180,E1 -11067.021,E2 -11067.021} C_VEL
LIN {X 0,Y 397.578,Z 194.957,A -85,B 0,C 180,E1 -11069.999,E2 -11069.999} C_VEL
LIN {X 0,Y 397.378,Z 194.989,A -85,B 0,C 180,E1 -11073.041,E2 -11073.041} C_VEL
LIN {X 0,Y 397.367,Z 194.983,A -85,B 0,C 180,E1 -11076.091,E2 -11076.091} C_VEL
LIN {X 0,Y 397.249,Z 195.002,A -85,B 0,C 180,E1 -11079.161,E2 -11079.161} C_VEL
LIN {X 0,Y 397.215,Z 195.003,A -85,B 0,C 180,E1 -11082.257,E2 -11082.257} C_VEL
LIN {X 0,Y 397.175,Z 195.009,A -85,B 0,C 180,E1 -11085.391,E2 -11085.391} C_VEL
LIN {X 0,Y 397.158,Z 195.014,A -85,B 0,C 180,E1 -11088.573,E2 -11088.573} C_VEL
LIN {X 0,Y 397.092,Z 195.018,A -85,B 0,C 180,E1 -11091.818,E2 -11091.818} C_VEL
LIN {X 0,Y 397.151,Z 195.012,A -85,B 0,C 180,E1 -11095.131,E2 -11095.131} C_VEL
LIN {X 0,Y 397.156,Z 195.01,A -85,B 0,C 180,E1 -11097.776,E2 -11097.776} C_VEL
LIN {X 0,Y 397.072,Z 195.024,A -85,B 0,C 180,E1 -11100.882,E2 -11100.882} C_VEL
LIN {X 0,Y 397.121,Z 195.021,A -85,B 0,C 180,E1 -11104.492,E2 -11104.492} C_VEL
LIN {X 0,Y 397.102,Z 195.021,A -85,B 0,C 180,E1 -11108.274,E2 -11108.274} C_VEL
LIN {X 0,Y 397.148,Z 195.013,A -85,B 0,C 180,E1 -11111.993,E2 -11111.993} C_VEL
LIN {X 0,Y 397.103,Z 195.017,A -85,B 0,C 180,E1 -11115.065,E2 -11115.065} C_VEL
LIN {X 0,Y 397.102,Z 195.02,A -85,B 0,C 180,E1 -11118.014,E2 -11118.014} C_VEL
LIN {X 0,Y 397.128,Z 195.013,A -85,B 0,C 180,E1 -11121.137,E2 -11121.137} C_VEL
LIN {X 0,Y 397.112,Z 195.019,A -85,B 0,C 180,E1 -11124.496,E2 -11124.496} C_VEL
LIN {X 0,Y 397.103,Z 195.02,A -85,B 0,C 180,E1 -11127.931,E2 -11127.931} C_VEL
LIN {X 0,Y 397.118,Z 195.015,A -85,B 0,C 180,E1 -11131.457,E2 -11131.457} C_VEL
LIN {X 0,Y 397.144,Z 195.014,A -85,B 0,C 180,E1 -11134.488,E2 -11134.488} C_VEL
LIN {X 0,Y 397.1,Z 195.016,A -85,B 0,C 180,E1 -11137.086,E2 -11137.086} C_VEL
LIN {X 0,Y 397.139,Z 195.014,A -85,B 0,C 180,E1 -11140.353,E2 -11140.353} C_VEL
LIN {X 0,Y 397.162,Z 195.012,A -85,B 0,C 180,E1 -11143.554,E2 -11143.554} C_VEL
LIN {X 0,Y 397.22,Z 195.002,A -85,B 0,C 180,E1 -11146.703,E2 -11146.703} C_VEL
LIN {X 0,Y 397.21,Z 195.01,A -85,B 0,C 180,E1 -11149.809,E2 -11149.809} C_VEL
LIN {X 0,Y 397.344,Z 194.986,A -85,B 0,C 180,E1 -11152.888,E2 -11152.888} C_VEL
LIN {X 0,Y 397.246,Z 194.999,A -85,B 0,C 180,E1 -11154.926,E2 -11154.926} C_VEL
LIN {X 0,Y 397.44,Z 194.978,A -85,B 0,C 180,E1 -11157.974,E2 -11157.974} C_VEL
LIN {X 0,Y 397.572,Z 194.961,A -85,B 0,C 180,E1 -11160,E2 -11160} C_VEL
LIN {X 0,Y 397.368,Z 194.984,A -85,B 0,C 180,E1 -11163.042,E2 -11163.042} C_VEL
LIN {X 0,Y 397.355,Z 194.987,A -85,B 0,C 180,E1 -11167.112,E2 -11167.112} C_VEL
LIN {X 0,Y 397.21,Z 195.004,A -85,B 0,C 180,E1 -11170.192,E2 -11170.192} C_VEL
LIN {X 0,Y 397.219,Z 195.007,A -85,B 0,C 180,E1 -11173.322,E2 -11173.322} C_VEL
LIN {X 0,Y 397.175,Z 195.011,A -85,B 0,C 180,E1 -11177.156,E2 -11177.156} C_VEL
LIN {X 0,Y 397.102,Z 195.017,A -85,B 0,C 180,E1 -11180.73,E2 -11180.73} C_VEL
LIN {X 0,Y 397.126,Z 195.014,A -85,B 0,C 180,E1 -11184.019,E2 -11184.019} C_VEL
LIN {X 0,Y 397.188,Z 195.011,A -85,B 0,C 180,E1 -11187.391,E2 -11187.391} C_VEL
LIN {X 0,Y 397.073,Z 195.023,A -85,B 0,C 180,E1 -11190.883,E2 -11190.883} C_VEL
LIN {X 0,Y 397.119,Z 195.015,A -85,B 0,C 180,E1 -11194.494,E2 -11194.494} C_VEL
LIN {X 0,Y 397.096,Z 195.017,A -85,B 0,C 180,E1 -11198.276,E2 -11198.276} C_VEL
LIN {X 0,Y 397.084,Z 195.024,A -85,B 0,C 180,E1 -11200.91,E2 -11200.91} C_VEL
LIN {X 0,Y 397.097,Z 195.018,A -85,B 0,C 180,E1 -11203.65,E2 -11203.65} C_VEL
LIN {X 0,Y 397.097,Z 195.019,A -85,B 0,C 180,E1 -11206.522,E2 -11206.522} C_VEL
LIN {X 0,Y 397.11,Z 195.017,A -85,B 0,C 180,E1 -11210.424,E2 -11210.424} C_VEL
LIN {X 0,Y 397.106,Z 195.017,A -85,B 0,C 180,E1 -11214.266,E2 -11214.266} C_VEL
LIN {X 0,Y 397.113,Z 195.022,A -85,B 0,C 180,E1 -11216.728,E2 -11216.728} C_VEL
LIN {X 0,Y 397.167,Z 195.202,A -85,B 0,C 180,E1 -11219.841,E2 -11219.841} C_VEL
LIN {X 0,Y 400.986,Z 211.976,A -85,B 0,C 180,E1 -11222.891,E2 -11222.891} C_VEL
LIN {X 0,Y 402.014,Z 217.576,A -85,B 0,C 180,E1 -11223.862,E2 -11223.862} C_VEL
LIN {X 0,Y 400.606,Z 235.803,A -85,B 0,C 180,E1 -11226.752,E2 -11226.752} C_VEL
LIN {X 0,Y 399.021,Z 259.294,A -85,B 0,C 180,E1 -11230.45,E2 -11230.45} C_VEL
LIN {X 0,Y 398.845,Z 262.689,A -85,B 0,C 180,E1 -11230.943,E2 -11230.943} C_VEL
LIN {X 0,Y 401.465,Z 289.249,A -85,B 0,C 180,E1 -11231.601,E2 -11231.601} C_VEL
LIN {X 0,Y 400.406,Z 369.838,A -85,B 0,C 180,E1 -11233.199,E2 -11233.199} C_VEL
LIN {X 0,Y 399.904,Z 383.153,A -85,B 0,C 180,E1 -11233.67,E2 -11233.67} C_VEL
LIN {X 0,Y 399.311,Z 395.23,A -85,B 0,C 180,E1 -11234.301,E2 -11234.301} C_VEL
LIN {X 0,Y 398.575,Z 407.739,A -85,B 0,C 180,E1 -11235.187,E2 -11235.187} C_VEL
LIN {X 0,Y 397.907,Z 418.172,A -85,B 0,C 180,E1 -11236.133,E2 -11236.133} C_VEL
LIN {X 0,Y 397.458,Z 427.899,A -85,B 0,C 180,E1 -11237.231,E2 -11237.231} C_VEL
LIN {X 0,Y 396.89,Z 435.423,A -85,B 0,C 180,E1 -11238.251,E2 -11238.251} C_VEL
LIN {X 0,Y 396.484,Z 443.276,A -85,B 0,C 180,E1 -11239.533,E2 -11239.533} C_VEL
LIN {X 0,Y 396.174,Z 450.915,A -85,B 0,C 180,E1 -11241.071,E2 -11241.071} C_VEL
LIN {X 0,Y 396.101,Z 456.086,A -85,B 0,C 180,E1 -11242.354,E2 -11242.354} C_VEL
LIN {X 0,Y 396.078,Z 461.044,A -85,B 0,C 180,E1 -11243.889,E2 -11243.889} C_VEL
LIN {X 0,Y 396.001,Z 464.781,A -85,B 0,C 180,E1 -11245.42,E2 -11245.42} C_VEL
LIN {X 0,Y 396.184,Z 467.443,A -85,B 0,C 180,E1 -11246.95,E2 -11246.95} C_VEL
LIN {X 0,Y 396.188,Z 468.651,A -85,B 0,C 180,E1 -11247.968,E2 -11247.968} C_VEL
LIN {X 0,Y 396.101,Z 469.374,A -85,B 0,C 180,E1 -11248.984,E2 -11248.984} C_VEL
LIN {X 0,Y 396.093,Z 469.668,A -85,B 0,C 180,E1 -11250.001,E2 -11250.001} C_VEL
LIN {X 0,Y 396.102,Z 469.55,A -85,B 0,C 180,E1 -11251.017,E2 -11251.017} C_VEL
LIN {X 0,Y 396.184,Z 469.003,A -85,B 0,C 180,E1 -11252.034,E2 -11252.034} C_VEL
LIN {X 0,Y 396.144,Z 467.982,A -85,B 0,C 180,E1 -11253.052,E2 -11253.052} C_VEL
LIN {X 0,Y 396.022,Z 466.538,A -85,B 0,C 180,E1 -11254.071,E2 -11254.071} C_VEL
LIN {X 0,Y 396.007,Z 463.52,A -85,B 0,C 180,E1 -11255.602,E2 -11255.602} C_VEL
LIN {X 0,Y 396.092,Z 459.414,A -85,B 0,C 180,E1 -11257.135,E2 -11257.135} C_VEL
LIN {X 0,Y 396.169,Z 453.089,A -85,B 0,C 180,E1 -11258.93,E2 -11258.93} C_VEL
LIN {X 0,Y 396.496,Z 446.154,A -85,B 0,C 180,E1 -11260.468,E2 -11260.468} C_VEL
LIN {X 0,Y 397.102,Z 437.56,A -85,B 0,C 180,E1 -11262.003,E2 -11262.003} C_VEL
LIN {X 0,Y 397.874,Z 427.537,A -85,B 0,C 180,E1 -11263.427,E2 -11263.427} C_VEL
LIN {X 0,Y 398.647,Z 416.629,A -85,B 0,C 180,E1 -11264.681,E2 -11264.681} C_VEL
LIN {X 0,Y 399.602,Z 405.44,A -85,B 0,C 180,E1 -11265.689,E2 -11265.689} C_VEL
LIN {X 0,Y 400.572,Z 392.928,A -85,B 0,C 180,E1 -11266.566,E2 -11266.566} C_VEL
LIN {X 0,Y 401.314,Z 380.889,A -85,B 0,C 180,E1 -11267.189,E2 -11267.189} C_VEL
LIN {X 0,Y 401.959,Z 367.772,A -85,B 0,C 180,E1 -11267.653,E2 -11267.653} C_VEL
LIN {X 0,Y 403.329,Z 288.508,A -85,B 0,C 180,E1 -11269.307,E2 -11269.307} C_VEL
LIN {X 0,Y 400.657,Z 265.615,A -85,B 0,C 180,E1 -11269.99,E2 -11269.99} C_VEL
LIN {X 0,Y 399.882,Z 260.522,A -85,B 0,C 180,E1 -11270.174,E2 -11270.174} C_VEL
LIN {X 0,Y 401.544,Z 237.078,A -85,B 0,C 180,E1 -11273.739,E2 -11273.739} C_VEL
LIN {X 0,Y 402.976,Z 218.805,A -85,B 0,C 180,E1 -11276.595,E2 -11276.595} C_VEL
LIN {X 0,Y 400.565,Z 207.436,A -85,B 0,C 180,E1 -11278.685,E2 -11278.685} C_VEL
LIN {X 0,Y 397.131,Z 195.26,A -85,B 0,C 180,E1 -11281.137,E2 -11281.137} C_VEL
LIN {X 0,Y 397.118,Z 195.021,A -85,B 0,C 180,E1 -11283.273,E2 -11283.273} C_VEL
LIN {X 0,Y 397.111,Z 195.02,A -85,B 0,C 180,E1 -11285.735,E2 -11285.735} C_VEL
LIN {X 0,Y 397.096,Z 195.023,A -85,B 0,C 180,E1 -11288.855,E2 -11288.855} C_VEL
LIN {X 0,Y 397.06,Z 195.026,A -85,B 0,C 180,E1 -11292.269,E2 -11292.269} C_VEL
LIN {X 0,Y 397.09,Z 195.024,A -85,B 0,C 180,E1 -11295.069,E2 -11295.069} C_VEL
LIN {X 0,Y 397.065,Z 195.021,A -85,B 0,C 180,E1 -11298.022,E2 -11298.022} C_VEL
LIN {X 0,Y 397.129,Z 195.018,A -85,B 0,C 180,E1 -11301.139,E2 -11301.139} C_VEL
LIN {X 0,Y 397.122,Z 195.016,A -85,B 0,C 180,E1 -11304.497,E2 -11304.497} C_VEL
LIN {X 0,Y 397.081,Z 195.022,A -85,B 0,C 180,E1 -11307.928,E2 -11307.928} C_VEL
LIN {X 0,Y 397.125,Z 195.017,A -85,B 0,C 180,E1 -11311.456,E2 -11311.456} C_VEL
LIN {X 0,Y 397.155,Z 195.015,A -85,B 0,C 180,E1 -11314.487,E2 -11314.487} C_VEL
LIN {X 0,Y 397.111,Z 195.017,A -85,B 0,C 180,E1 -11317.085,E2 -11317.085} C_VEL
LIN {X 0,Y 397.15,Z 195.017,A -85,B 0,C 180,E1 -11320.352,E2 -11320.352} C_VEL
LIN {X 0,Y 397.168,Z 195.012,A -85,B 0,C 180,E1 -11323.553,E2 -11323.553} C_VEL
LIN {X 0,Y 397.231,Z 195.007,A -85,B 0,C 180,E1 -11326.702,E2 -11326.702} C_VEL
LIN {X 0,Y 397.219,Z 195.008,A -85,B 0,C 180,E1 -11329.809,E2 -11329.809} C_VEL
LIN {X 0,Y 397.319,Z 194.995,A -85,B 0,C 180,E1 -11332.887,E2 -11332.887} C_VEL
LIN {X 0,Y 397.257,Z 195.215,A -85,B 0,C 180,E1 -11335.465,E2 -11335.465} C_VEL
LIN {X 0,Y 399.927,Z 205.066,A -85,B 0,C 180,E1 -11337.733,E2 -11337.733} C_VEL
LIN {X 0,Y 400.574,Z 209.817,A -85,B 0,C 180,E1 -11338.743,E2 -11338.743} C_VEL
LIN {X 0,Y 399.929,Z 226.497,A -85,B 0,C 180,E1 -11342.014,E2 -11342.014} C_VEL
LIN {X 0,Y 399.881,Z 231.013,A -85,B 0,C 180,E1 -11342.833,E2 -11342.833} C_VEL
LIN {X 0,Y 403.417,Z 247.125,A -85,B 0,C 180,E1 -11343.497,E2 -11343.497} C_VEL
LIN {X 0,Y 403.504,Z 252.203,A -85,B 0,C 180,E1 -11343.634,E2 -11343.634} C_VEL
LIN {X 0,Y 401.894,Z 315.389,A -85,B 0,C 180,E1 -11345.173,E2 -11345.173} C_VEL
LIN {X 0,Y 401.595,Z 327.127,A -85,B 0,C 180,E1 -11345.649,E2 -11345.649} C_VEL
LIN {X 0,Y 401.1,Z 338.076,A -85,B 0,C 180,E1 -11346.287,E2 -11346.287} C_VEL
LIN {X 0,Y 400.591,Z 348.056,A -85,B 0,C 180,E1 -11347.054,E2 -11347.054} C_VEL
LIN {X 0,Y 399.901,Z 358.392,A -85,B 0,C 180,E1 -11348.082,E2 -11348.082} C_VEL
LIN {X 0,Y 399.286,Z 366.642,A -85,B 0,C 180,E1 -11349.114,E2 -11349.114} C_VEL
LIN {X 0,Y 398.599,Z 374.897,A -85,B 0,C 180,E1 -11350.412,E2 -11350.412} C_VEL
LIN {X 0,Y 398.018,Z 381.454,A -85,B 0,C 180,E1 -11351.715,E2 -11351.715} C_VEL
LIN {X 0,Y 397.44,Z 387.571,A -85,B 0,C 180,E1 -11353.29,E2 -11353.29} C_VEL
LIN {X 0,Y 396.974,Z 392.053,A -85,B 0,C 180,E1 -11354.874,E2 -11354.874} C_VEL
LIN {X 0,Y 396.691,Z 395.126,A -85,B 0,C 180,E1 -11356.467,E2 -11356.467} C_VEL
LIN {X 0,Y 396.509,Z 396.416,A -85,B 0,C 180,E1 -11357.536,E2 -11357.536} C_VEL
LIN {X 0,Y 396.36,Z 397.137,A -85,B 0,C 180,E1 -11358.612,E2 -11358.612} C_VEL
LIN {X 0,Y 396.271,Z 397.227,A -85,B 0,C 180,E1 -11359.952,E2 -11359.952} C_VEL
LIN {X 0,Y 396.237,Z 396.84,A -85,B 0,C 180,E1 -11360.777,E2 -11360.777} C_VEL
LIN {X 0,Y 396.256,Z 395.805,A -85,B 0,C 180,E1 -11361.867,E2 -11361.867} C_VEL
LIN {X 0,Y 396.424,Z 393.104,A -85,B 0,C 180,E1 -11363.508,E2 -11363.508} C_VEL
LIN {X 0,Y 396.637,Z 388.851,A -85,B 0,C 180,E1 -11365.166,E2 -11365.166} C_VEL
LIN {X 0,Y 396.885,Z 383.991,A -85,B 0,C 180,E1 -11366.559,E2 -11366.559} C_VEL
LIN {X 0,Y 397.282,Z 376.943,A -85,B 0,C 180,E1 -11368.097,E2 -11368.097} C_VEL
LIN {X 0,Y 397.669,Z 369.511,A -85,B 0,C 180,E1 -11369.368,E2 -11369.368} C_VEL
LIN {X 0,Y 398.193,Z 360.804,A -85,B 0,C 180,E1 -11370.556,E2 -11370.556} C_VEL
LIN {X 0,Y 398.639,Z 350.802,A -85,B 0,C 180,E1 -11371.633,E2 -11371.633} C_VEL
LIN {X 0,Y 399.081,Z 341.085,A -85,B 0,C 180,E1 -11372.459,E2 -11372.459} C_VEL
LIN {X 0,Y 399.475,Z 329.601,A -85,B 0,C 180,E1 -11373.201,E2 -11373.201} C_VEL
LIN {X 0,Y 399.698,Z 317.736,A -85,B 0,C 180,E1 -11373.746,E2 -11373.746} C_VEL
LIN {X 0,Y 399.897,Z 305.141,A -85,B 0,C 180,E1 -11374.106,E2 -11374.106} C_VEL
LIN {X 0,Y 400.748,Z 244.978,A -85,B 0,C 180,E1 -11375.399,E2 -11375.399} C_VEL
LIN {X 0,Y 398.153,Z 229.171,A -85,B 0,C 180,E1 -11375.864,E2 -11375.864} C_VEL
LIN {X 0,Y 398.169,Z 226.983,A -85,B 0,C 180,E1 -11376.248,E2 -11376.248} C_VEL
LIN {X 0,Y 398.635,Z 212.446,A -85,B 0,C 180,E1 -11379.396,E2 -11379.396} C_VEL
LIN {X 0,Y 398.889,Z 205.067,A -85,B 0,C 180,E1 -11381.017,E2 -11381.017} C_VEL
LIN {X 0,Y 397.573,Z 197.38,A -85,B 0,C 180,E1 -11382.81,E2 -11382.81} C_VEL
LIN {X 0,Y 397.112,Z 195.058,A -85,B 0,C 180,E1 -11383.434,E2 -11383.434} C_VEL
LIN {X 0,Y 397.101,Z 195.021,A -85,B 0,C 180,E1 -11386.52,E2 -11386.52} C_VEL
LIN {X 0,Y 397.111,Z 195.016,A -85,B 0,C 180,E1 -11390.422,E2 -11390.422} C_VEL
LIN {X 0,Y 397.107,Z 195.017,A -85,B 0,C 180,E1 -11394.265,E2 -11394.265} C_VEL
LIN {X 0,Y 397.113,Z 195.015,A -85,B 0,C 180,E1 -11396.727,E2 -11396.727} C_VEL
LIN {X 0,Y 397.123,Z 195.014,A -85,B 0,C 180,E1 -11400.295,E2 -11400.295} C_VEL
LIN {X 0,Y 397.193,Z 195.005,A -85,B 0,C 180,E1 -11402.609,E2 -11402.609} C_VEL
LIN {X 0,Y 397.132,Z 195.014,A -85,B 0,C 180,E1 -11405.981,E2 -11405.981} C_VEL
LIN {X 0,Y 397.137,Z 195.015,A -85,B 0,C 180,E1 -11409.704,E2 -11409.704} C_VEL
LIN {X 0,Y 397.18,Z 195.008,A -85,B 0,C 180,E1 -11412.844,E2 -11412.844} C_VEL
LIN {X 0,Y 397.226,Z 195.002,A -85,B 0,C 180,E1 -11416.702,E2 -11416.702} C_VEL
LIN {X 0,Y 397.216,Z 195.003,A -85,B 0,C 180,E1 -11419.808,E2 -11419.808} C_VEL
LIN {X 0,Y 397.362,Z 194.987,A -85,B 0,C 180,E1 -11422.888,E2 -11422.888} C_VEL
LIN {X 0,Y 397.253,Z 195.002,A -85,B 0,C 180,E1 -11424.924,E2 -11424.924} C_VEL
LIN {X 0,Y 397.379,Z 194.986,A -85,B 0,C 180,E1 -11427.021,E2 -11427.021} C_VEL
LIN {X 0,Y 396.721,Z 195.065,A -85,B 0,C 180,E1 -11427.869,E2 -11427.869} C_VEL
LIN {X 0,Y 393.854,Z 195.426,A -85,B 0,C 180,E1 -11429.247,E2 -11429.247} C_VEL
LIN {X 0,Y 391.439,Z 195.728,A -85,B 0,C 180,E1 -11430.361,E2 -11430.361} C_VEL
LIN {X 0,Y 390.432,Z 195.852,A -85,B 0,C 180,E1 -11431.222,E2 -11431.222} C_VEL
LIN {X 0,Y 390.366,Z 195.857,A -85,B 0,C 180,E1 -11431.513,E2 -11431.513} C_VEL
LIN {X 0,Y 390.111,Z 195.887,A -85,B 0,C 180,E1 -11434.132,E2 -11434.132} C_VEL
LIN {X 0,Y 390.321,Z 195.861,A -85,B 0,C 180,E1 -11436.201,E2 -11436.201} C_VEL
LIN {X 0,Y 390.201,Z 195.879,A -85,B 0,C 180,E1 -11439.328,E2 -11439.328} C_VEL
LIN {X 0,Y 390.19,Z 195.879,A -85,B 0,C 180,E1 -11443.438,E2 -11443.438} C_VEL
LIN {X 0,Y 390.144,Z 195.885,A -85,B 0,C 180,E1 -11447.307,E2 -11447.307} C_VEL
LIN {X 0,Y 390.082,Z 195.894,A -85,B 0,C 180,E1 -11450.469,E2 -11450.469} C_VEL
LIN {X 0,Y 390.084,Z 195.891,A -85,B 0,C 180,E1 -11453.35,E2 -11453.35} C_VEL
LIN {X 0,Y 390.108,Z 195.893,A -85,B 0,C 180,E1 -11456.767,E2 -11456.767} C_VEL
LIN {X 0,Y 390.033,Z 195.9,A -85,B 0,C 180,E1 -11460.299,E2 -11460.299} C_VEL
LIN {X 0,Y 390.084,Z 195.892,A -85,B 0,C 180,E1 -11464.029,E2 -11464.029} C_VEL
LIN {X 0,Y 390.04,Z 195.897,A -85,B 0,C 180,E1 -11467.779,E2 -11467.779} C_VEL
LIN {X 0,Y 390.075,Z 195.894,A -85,B 0,C 180,E1 -11470.825,E2 -11470.825} C_VEL
LIN {X 0,Y 390.094,Z 195.891,A -85,B 0,C 180,E1 -11473.893,E2 -11473.893} C_VEL
LIN {X 0,Y 390.073,Z 195.892,A -85,B 0,C 180,E1 -11477.619,E2 -11477.619} C_VEL
LIN {X 0,Y 390.086,Z 195.891,A -85,B 0,C 180,E1 -11480.908,E2 -11480.908} C_VEL
LIN {X 0,Y 390.077,Z 195.893,A -85,B 0,C 180,E1 -11484.793,E2 -11484.793} C_VEL
LIN {X 0,Y 390.041,Z 195.899,A -85,B 0,C 180,E1 -11488.498,E2 -11488.498} C_VEL
LIN {X 0,Y 390.109,Z 195.894,A -85,B 0,C 180,E1 -11492.07,E2 -11492.07} C_VEL
LIN {X 0,Y 390.071,Z 195.894,A -85,B 0,C 180,E1 -11495.519,E2 -11495.519} C_VEL
LIN {X 0,Y 390.047,Z 195.895,A -85,B 0,C 180,E1 -11498.878,E2 -11498.878} C_VEL
LIN {X 0,Y 390.12,Z 195.891,A -85,B 0,C 180,E1 -11502.167,E2 -11502.167} C_VEL
LIN {X 0,Y 390.138,Z 195.886,A -85,B 0,C 180,E1 -11505.393,E2 -11505.393} C_VEL
LIN {X 0,Y 390.14,Z 195.884,A -85,B 0,C 180,E1 -11508.571,E2 -11508.571} C_VEL
LIN {X 0,Y 390.299,Z 195.868,A -85,B 0,C 180,E1 -11512.032,E2 -11512.032} C_VEL
LIN {X 0,Y 390.218,Z 195.874,A -85,B 0,C 180,E1 -11514.834,E2 -11514.834} C_VEL
LIN {X 0,Y 390.409,Z 195.854,A -85,B 0,C 180,E1 -11517.937,E2 -11517.937} C_VEL
LIN {X 0,Y 390.542,Z 195.837,A -85,B 0,C 180,E1 -11520,E2 -11520} C_VEL
LIN {X 0,Y 390.302,Z 195.865,A -85,B 0,C 180,E1 -11523.097,E2 -11523.097} C_VEL
LIN {X 0,Y 390.319,Z 195.862,A -85,B 0,C 180,E1 -11526.203,E2 -11526.203} C_VEL
LIN {X 0,Y 390.307,Z 195.863,A -85,B 0,C 180,E1 -11528.283,E2 -11528.283} C_VEL
LIN {X 0,Y 390.163,Z 195.881,A -85,B 0,C 180,E1 -11532.484,E2 -11532.484} C_VEL
LIN {X 0,Y 390.132,Z 195.889,A -85,B 0,C 180,E1 -11535.678,E2 -11535.678} C_VEL
LIN {X 0,Y 390.099,Z 195.891,A -85,B 0,C 180,E1 -11538.923,E2 -11538.923} C_VEL
LIN {X 0,Y 390.04,Z 195.896,A -85,B 0,C 180,E1 -11542.235,E2 -11542.235} C_VEL
LIN {X 0,Y 390.113,Z 195.889,A -85,B 0,C 180,E1 -11545.744,E2 -11545.744} C_VEL
LIN {X 0,Y 390.053,Z 195.9,A -85,B 0,C 180,E1 -11549.11,E2 -11549.11} C_VEL
LIN {X 0,Y 390.037,Z 195.899,A -85,B 0,C 180,E1 -11552.723,E2 -11552.723} C_VEL
LIN {X 0,Y 390.05,Z 195.895,A -85,B 0,C 180,E1 -11555.826,E2 -11555.826} C_VEL
LIN {X 0,Y 390.064,Z 195.898,A -85,B 0,C 180,E1 -11559.219,E2 -11559.219} C_VEL
LIN {X 0,Y 390.038,Z 195.897,A -85,B 0,C 180,E1 -11562.375,E2 -11562.375} C_VEL
LIN {X 0,Y 390.041,Z 195.899,A -85,B 0,C 180,E1 -11565.355,E2 -11565.355} C_VEL
LIN {X 0,Y 390.024,Z 195.898,A -85,B 0,C 180,E1 -11568.187,E2 -11568.187} C_VEL
LIN {X 0,Y 390.085,Z 195.897,A -85,B 0,C 180,E1 -11570.908,E2 -11570.908} C_VEL
LIN {X 0,Y 390.083,Z 195.897,A -85,B 0,C 180,E1 -11574.794,E2 -11574.794} C_VEL
LIN {X 0,Y 390.025,Z 195.904,A -85,B 0,C 180,E1 -11578.497,E2 -11578.497} C_VEL
LIN {X 0,Y 390.104,Z 196.137,A -85,B 0,C 180,E1 -11579.576,E2 -11579.576} C_VEL
LIN {X 0,Y 394.119,Z 213.683,A -85,B 0,C 180,E1 -11582.814,E2 -11582.814} C_VEL
LIN {X 0,Y 394.99,Z 218.053,A -85,B 0,C 180,E1 -11583.589,E2 -11583.589} C_VEL
LIN {X 0,Y 394.436,Z 227.639,A -85,B 0,C 180,E1 -11585.149,E2 -11585.149} C_VEL
LIN {X 0,Y 392.443,Z 253.405,A -85,B 0,C 180,E1 -11589.288,E2 -11589.288} C_VEL
LIN {X 0,Y 391.85,Z 262.273,A -85,B 0,C 180,E1 -11590.677,E2 -11590.677} C_VEL
LIN {X 0,Y 392.876,Z 273.718,A -85,B 0,C 180,E1 -11590.989,E2 -11590.989} C_VEL
LIN {X 0,Y 394.557,Z 290.146,A -85,B 0,C 180,E1 -11591.387,E2 -11591.387} C_VEL
LIN {X 0,Y 393.46,Z 369.223,A -85,B 0,C 180,E1 -11592.994,E2 -11592.994} C_VEL
LIN {X 0,Y 392.936,Z 382.549,A -85,B 0,C 180,E1 -11593.472,E2 -11593.472} C_VEL
LIN {X 0,Y 392.296,Z 395.142,A -85,B 0,C 180,E1 -11594.146,E2 -11594.146} C_VEL
LIN {X 0,Y 391.536,Z 407.553,A -85,B 0,C 180,E1 -11595.048,E2 -11595.048} C_VEL
LIN {X 0,Y 390.814,Z 418.748,A -85,B 0,C 180,E1 -11596.1,E2 -11596.1} C_VEL
LIN {X 0,Y 390.306,Z 428.556,A -85,B 0,C 180,E1 -11597.258,E2 -11597.258} C_VEL
LIN {X 0,Y 389.704,Z 437.551,A -85,B 0,C 180,E1 -11598.559,E2 -11598.559} C_VEL
LIN {X 0,Y 389.279,Z 444.939,A -85,B 0,C 180,E1 -11599.863,E2 -11599.863} C_VEL
LIN {X 0,Y 389.092,Z 452.139,A -85,B 0,C 180,E1 -11601.431,E2 -11601.431} C_VEL
LIN {X 0,Y 389.027,Z 458.652,A -85,B 0,C 180,E1 -11603.258,E2 -11603.258} C_VEL
LIN {X 0,Y 388.976,Z 462.848,A -85,B 0,C 180,E1 -11604.818,E2 -11604.818} C_VEL
LIN {X 0,Y 388.973,Z 465.002,A -85,B 0,C 180,E1 -11605.856,E2 -11605.856} C_VEL
LIN {X 0,Y 389.109,Z 466.68,A -85,B 0,C 180,E1 -11606.895,E2 -11606.895} C_VEL
LIN {X 0,Y 389.139,Z 467.911,A -85,B 0,C 180,E1 -11607.931,E2 -11607.931} C_VEL
LIN {X 0,Y 389.049,Z 468.676,A -85,B 0,C 180,E1 -11608.966,E2 -11608.966} C_VEL
LIN {X 0,Y 389.037,Z 468.99,A -85,B 0,C 180,E1 -11610.001,E2 -11610.001} C_VEL
LIN {X 0,Y 389.05,Z 468.889,A -85,B 0,C 180,E1 -11611.036,E2 -11611.036} C_VEL
LIN {X 0,Y 389.116,Z 468.371,A -85,B 0,C 180,E1 -11612.071,E2 -11612.071} C_VEL
LIN {X 0,Y 389.072,Z 467.37,A -85,B 0,C 180,E1 -11613.107,E2 -11613.107} C_VEL
LIN {X 0,Y 388.932,Z 465.935,A -85,B 0,C 180,E1 -11614.146,E2 -11614.146} C_VEL
LIN {X 0,Y 388.91,Z 462.943,A -85,B 0,C 180,E1 -11615.705,E2 -11615.705} C_VEL
LIN {X 0,Y 389.013,Z 458.863,A -85,B 0,C 180,E1 -11617.266,E2 -11617.266} C_VEL
LIN {X 0,Y 389.096,Z 453.584,A -85,B 0,C 180,E1 -11618.832,E2 -11618.832} C_VEL
LIN {X 0,Y 389.362,Z 446.963,A -85,B 0,C 180,E1 -11620.4,E2 -11620.4} C_VEL
LIN {X 0,Y 389.995,Z 438.699,A -85,B 0,C 180,E1 -11621.961,E2 -11621.961} C_VEL
LIN {X 0,Y 390.697,Z 430.284,A -85,B 0,C 180,E1 -11623.259,E2 -11623.259} C_VEL
LIN {X 0,Y 391.475,Z 419.991,A -85,B 0,C 180,E1 -11624.557,E2 -11624.557} C_VEL
LIN {X 0,Y 392.487,Z 408.346,A -85,B 0,C 180,E1 -11625.714,E2 -11625.714} C_VEL
LIN {X 0,Y 393.496,Z 396.906,A -85,B 0,C 180,E1 -11626.605,E2 -11626.605} C_VEL
LIN {X 0,Y 394.344,Z 383.84,A -85,B 0,C 180,E1 -11627.369,E2 -11627.369} C_VEL
LIN {X 0,Y 395.135,Z 370.755,A -85,B 0,C 180,E1 -11627.901,E2 -11627.901} C_VEL
LIN {X 0,Y 395.568,Z 355.068,A -85,B 0,C 180,E1 -11628.283,E2 -11628.283} C_VEL
LIN {X 0,Y 396.732,Z 288.668,A -85,B 0,C 180,E1 -11629.699,E2 -11629.699} C_VEL
LIN {X 0,Y 394.153,Z 266.595,A -85,B 0,C 180,E1 -11630.384,E2 -11630.384} C_VEL
LIN {X 0,Y 393.165,Z 260.054,A -85,B 0,C 180,E1 -11630.622,E2 -11630.622} C_VEL
LIN {X 0,Y 395.221,Z 233.682,A -85,B 0,C 180,E1 -11634.733,E2 -11634.733} C_VEL
LIN {X 0,Y 396.269,Z 220.744,A -85,B 0,C 180,E1 -11636.796,E2 -11636.796} C_VEL
LIN {X 0,Y 393.786,Z 209.031,A -85,B 0,C 180,E1 -11639.011,E2 -11639.011} C_VEL
LIN {X 0,Y 390.19,Z 196.569,A -85,B 0,C 180,E1 -11641.6,E2 -11641.6} C_VEL
LIN {X 0,Y 390.052,Z 195.952,A -85,B 0,C 180,E1 -11641.834,E2 -11641.834} C_VEL
LIN {X 0,Y 390.088,Z 195.897,A -85,B 0,C 180,E1 -11645.207,E2 -11645.207} C_VEL
LIN {X 0,Y 390.061,Z 195.899,A -85,B 0,C 180,E1 -11649.096,E2 -11649.096} C_VEL
LIN {X 0,Y 390.035,Z 195.901,A -85,B 0,C 180,E1 -11652.372,E2 -11652.372} C_VEL
LIN {X 0,Y 390.047,Z 195.9,A -85,B 0,C 180,E1 -11655.354,E2 -11655.354} C_VEL
LIN {X 0,Y 390.03,Z 195.898,A -85,B 0,C 180,E1 -11658.186,E2 -11658.186} C_VEL
LIN {X 0,Y 390.09,Z 195.896,A -85,B 0,C 180,E1 -11660.907,E2 -11660.907} C_VEL
LIN {X 0,Y 390.087,Z 195.894,A -85,B 0,C 180,E1 -11664.793,E2 -11664.793} C_VEL
LIN {X 0,Y 390.026,Z 195.9,A -85,B 0,C 180,E1 -11668.495,E2 -11668.495} C_VEL
LIN {X 0,Y 390.12,Z 195.89,A -85,B 0,C 180,E1 -11672.07,E2 -11672.07} C_VEL
LIN {X 0,Y 390.082,Z 195.893,A -85,B 0,C 180,E1 -11675.519,E2 -11675.519} C_VEL
LIN {X 0,Y 390.058,Z 195.897,A -85,B 0,C 180,E1 -11678.877,E2 -11678.877} C_VEL
LIN {X 0,Y 390.13,Z 195.891,A -85,B 0,C 180,E1 -11682.166,E2 -11682.166} C_VEL
LIN {X 0,Y 390.146,Z 195.887,A -85,B 0,C 180,E1 -11685.392,E2 -11685.392} C_VEL
LIN {X 0,Y 390.15,Z 195.888,A -85,B 0,C 180,E1 -11688.571,E2 -11688.571} C_VEL
LIN {X 0,Y 390.26,Z 195.875,A -85,B 0,C 180,E1 -11692.084,E2 -11692.084} C_VEL
LIN {X 0,Y 390.244,Z 196.037,A -85,B 0,C 180,E1 -11694.898,E2 -11694.898} C_VEL
LIN {X 0,Y 393.137,Z 206.713,A -85,B 0,C 180,E1 -11697.438,E2 -11697.438} C_VEL
LIN {X 0,Y 393.894,Z 211.149,A -85,B 0,C 180,E1 -11698.415,E2 -11698.415} C_VEL
LIN {X 0,Y 393.284,Z 225.533,A -85,B 0,C 180,E1 -11701.279,E2 -11701.279} C_VEL
LIN {X 0,Y 393.191,Z 231.23,A -85,B 0,C 180,E1 -11702.372,E2 -11702.372} C_VEL
LIN {X 0,Y 396.739,Z 247.369,A -85,B 0,C 180,E1 -11703.077,E2 -11703.077} C_VEL
LIN {X 0,Y 397.056,Z 250.724,A -85,B 0,C 180,E1 -11703.186,E2 -11703.186} C_VEL
LIN {X 0,Y 395.255,Z 315.703,A -85,B 0,C 180,E1 -11704.812,E2 -11704.812} C_VEL
LIN {X 0,Y 394.946,Z 327.425,A -85,B 0,C 180,E1 -11705.296,E2 -11705.296} C_VEL
LIN {X 0,Y 394.385,Z 339.337,A -85,B 0,C 180,E1 -11706.009,E2 -11706.009} C_VEL
LIN {X 0,Y 393.695,Z 350.585,A -85,B 0,C 180,E1 -11706.92,E2 -11706.92} C_VEL
LIN {X 0,Y 393,Z 360.54,A -85,B 0,C 180,E1 -11707.966,E2 -11707.966} C_VEL
LIN {X 0,Y 392.382,Z 368.481,A -85,B 0,C 180,E1 -11709.016,E2 -11709.016} C_VEL
LIN {X 0,Y 391.639,Z 376.533,A -85,B 0,C 180,E1 -11710.337,E2 -11710.337} C_VEL
LIN {X 0,Y 390.934,Z 384.017,A -85,B 0,C 180,E1 -11711.931,E2 -11711.931} C_VEL
LIN {X 0,Y 390.355,Z 389.635,A -85,B 0,C 180,E1 -11713.535,E2 -11713.535} C_VEL
LIN {X 0,Y 389.896,Z 393.721,A -85,B 0,C 180,E1 -11715.151,E2 -11715.151} C_VEL
LIN {X 0,Y 389.52,Z 396.689,A -85,B 0,C 180,E1 -11717.007,E2 -11717.007} C_VEL
LIN {X 0,Y 389.402,Z 397.457,A -85,B 0,C 180,E1 -11717.867,E2 -11717.867} C_VEL
LIN {X 0,Y 389.261,Z 397.961,A -85,B 0,C 180,E1 -11718.964,E2 -11718.964} C_VEL
LIN {X 0,Y 389.209,Z 397.831,A -85,B 0,C 180,E1 -11720.12,E2 -11720.12} C_VEL
LIN {X 0,Y 389.175,Z 397.165,A -85,B 0,C 180,E1 -11721.172,E2 -11721.172} C_VEL
LIN {X 0,Y 389.291,Z 394.793,A -85,B 0,C 180,E1 -11722.968,E2 -11722.968} C_VEL
LIN {X 0,Y 389.49,Z 391.381,A -85,B 0,C 180,E1 -11724.52,E2 -11724.52} C_VEL
LIN {X 0,Y 389.78,Z 386.102,A -85,B 0,C 180,E1 -11726.215,E2 -11726.215} C_VEL
LIN {X 0,Y 390.063,Z 380.186,A -85,B 0,C 180,E1 -11727.642,E2 -11727.642} C_VEL
LIN {X 0,Y 390.501,Z 372.578,A -85,B 0,C 180,E1 -11729.073,E2 -11729.073} C_VEL
LIN {X 0,Y 390.972,Z 363.881,A -85,B 0,C 180,E1 -11730.363,E2 -11730.363} C_VEL
LIN {X 0,Y 391.515,Z 353.962,A -85,B 0,C 180,E1 -11731.521,E2 -11731.521} C_VEL
LIN {X 0,Y 392.04,Z 342.719,A -85,B 0,C 180,E1 -11732.534,E2 -11732.534} C_VEL
LIN {X 0,Y 392.407,Z 332.089,A -85,B 0,C 180,E1 -11733.263,E2 -11733.263} C_VEL
LIN {X 0,Y 392.761,Z 320.007,A -85,B 0,C 180,E1 -11733.863,E2 -11733.863} C_VEL
LIN {X 0,Y 392.929,Z 306.905,A -85,B 0,C 180,E1 -11734.272,E2 -11734.272} C_VEL
LIN {X 0,Y 393.981,Z 246.657,A -85,B 0,C 180,E1 -11735.597,E2 -11735.597} C_VEL
LIN {X 0,Y 391.189,Z 229.544,A -85,B 0,C 180,E1 -11736.104,E2 -11736.104} C_VEL
LIN {X 0,Y 391.193,Z 227.878,A -85,B 0,C 180,E1 -11736.36,E2 -11736.36} C_VEL
LIN {X 0,Y 391.698,Z 212.315,A -85,B 0,C 180,E1 -11739.771,E2 -11739.771} C_VEL
LIN {X 0,Y 391.922,Z 206.173,A -85,B 0,C 180,E1 -11741.136,E2 -11741.136} C_VEL
LIN {X 0,Y 390.398,Z 197.619,A -85,B 0,C 180,E1 -11743.163,E2 -11743.163} C_VEL
LIN {X 0,Y 390.066,Z 195.931,A -85,B 0,C 180,E1 -11743.646,E2 -11743.646} C_VEL
LIN {X 0,Y 390.056,Z 195.898,A -85,B 0,C 180,E1 -11746.789,E2 -11746.789} C_VEL
LIN {X 0,Y 390.055,Z 195.899,A -85,B 0,C 180,E1 -11749.56,E2 -11749.56} C_VEL
LIN {X 0,Y 390.041,Z 195.896,A -85,B 0,C 180,E1 -11752.449,E2 -11752.449} C_VEL
LIN {X 0,Y 390.067,Z 195.896,A -85,B 0,C 180,E1 -11755.975,E2 -11755.975} C_VEL
LIN {X 0,Y 390.045,Z 195.899,A -85,B 0,C 180,E1 -11759.868,E2 -11759.868} C_VEL
LIN {X 0,Y 390.112,Z 195.891,A -85,B 0,C 180,E1 -11763.231,E2 -11763.231} C_VEL
LIN {X 0,Y 390.105,Z 195.889,A -85,B 0,C 180,E1 -11766.75,E2 -11766.75} C_VEL
LIN {X 0,Y 390.102,Z 195.89,A -85,B 0,C 180,E1 -11769.982,E2 -11769.982} C_VEL
LIN {X 0,Y 390.136,Z 195.89,A -85,B 0,C 180,E1 -11773.248,E2 -11773.248} C_VEL
LIN {X 0,Y 390.192,Z 195.878,A -85,B 0,C 180,E1 -11776.561,E2 -11776.561} C_VEL
LIN {X 0,Y 390.203,Z 195.877,A -85,B 0,C 180,E1 -11780.671,E2 -11780.671} C_VEL
LIN {X 0,Y 390.316,Z 195.864,A -85,B 0,C 180,E1 -11782.758,E2 -11782.758} C_VEL
LIN {X 0,Y 390.225,Z 195.876,A -85,B 0,C 180,E1 -11784.833,E2 -11784.833} C_VEL
LIN {X 0,Y 390.418,Z 195.849,A -85,B 0,C 180,E1 -11787.936,E2 -11787.936} C_VEL
LIN {X 0,Y 390.548,Z 195.833,A -85,B 0,C 180,E1 -11789.999,E2 -11789.999} C_VEL
LIN {X 0,Y 390.366,Z 195.857,A -85,B 0,C 180,E1 -11791.513,E2 -11791.513} C_VEL
LIN {X 0,Y 389.716,Z 195.938,A -85,B 0,C 180,E1 -11792.373,E2 -11792.373} C_VEL
LIN {X 0,Y 386.784,Z 196.302,A -85,B 0,C 180,E1 -11793.768,E2 -11793.768} C_VEL
LIN {X 0,Y 384.313,Z 196.615,A -85,B 0,C 180,E1 -11794.896,E2 -11794.896} C_VEL
LIN {X 0,Y 383.3,Z 196.736,A -85,B 0,C 180,E1 -11795.77,E2 -11795.77} C_VEL
LIN {X 0,Y 383.246,Z 196.742,A -85,B 0,C 180,E1 -11796.066,E2 -11796.066} C_VEL
LIN {X 0,Y 383.218,Z 196.747,A -85,B 0,C 180,E1 -11798.436,E2 -11798.436} C_VEL
LIN {X 0,Y 383.094,Z 196.762,A -85,B 0,C 180,E1 -11801.641,E2 -11801.641} C_VEL
LIN {X 0,Y 383.106,Z 196.766,A -85,B 0,C 180,E1 -11804.881,E2 -11804.881} C_VEL
LIN {X 0,Y 383.085,Z 196.763,A -85,B 0,C 180,E1 -11808.172,E2 -11808.172} C_VEL
LIN {X 0,Y 382.988,Z 196.775,A -85,B 0,C 180,E1 -11811.53,E2 -11811.53} C_VEL
LIN {X 0,Y 383.047,Z 196.771,A -85,B 0,C 180,E1 -11814.96,E2 -11814.96} C_VEL
LIN {X 0,Y 383.034,Z 196.774,A -85,B 0,C 180,E1 -11818.492,E2 -11818.492} C_VEL
LIN {X 0,Y 383.003,Z 196.775,A -85,B 0,C 180,E1 -11822.149,E2 -11822.149} C_VEL
LIN {X 0,Y 383.02,Z 196.776,A -85,B 0,C 180,E1 -11824.666,E2 -11824.666} C_VEL
LIN {X 0,Y 382.996,Z 196.775,A -85,B 0,C 180,E1 -11827.904,E2 -11827.904} C_VEL
LIN {X 0,Y 383.039,Z 196.768,A -85,B 0,C 180,E1 -11831.339,E2 -11831.339} C_VEL
LIN {X 0,Y 383.026,Z 196.776,A -85,B 0,C 180,E1 -11834.309,E2 -11834.309} C_VEL
LIN {X 0,Y 383.031,Z 196.769,A -85,B 0,C 180,E1 -11837.244,E2 -11837.244} C_VEL
LIN {X 0,Y 383.013,Z 196.777,A -85,B 0,C 180,E1 -11840.412,E2 -11840.412} C_VEL
LIN {X 0,Y 383.018,Z 196.775,A -85,B 0,C 180,E1 -11844.044,E2 -11844.044} C_VEL
LIN {X 0,Y 383.029,Z 196.773,A -85,B 0,C 180,E1 -11847.853,E2 -11847.853} C_VEL
LIN {X 0,Y 383.056,Z 196.769,A -85,B 0,C 180,E1 -11851.72,E2 -11851.72} C_VEL
LIN {X 0,Y 383.043,Z 196.768,A -85,B 0,C 180,E1 -11855.04,E2 -11855.04} C_VEL
LIN {X 0,Y 382.984,Z 196.777,A -85,B 0,C 180,E1 -11858.469,E2 -11858.469} C_VEL
LIN {X 0,Y 383.081,Z 196.768,A -85,B 0,C 180,E1 -11861.828,E2 -11861.828} C_VEL
LIN {X 0,Y 383.104,Z 196.76,A -85,B 0,C 180,E1 -11865.119,E2 -11865.119} C_VEL
LIN {X 0,Y 383.09,Z 196.764,A -85,B 0,C 180,E1 -11868.358,E2 -11868.358} C_VEL
LIN {X 0,Y 383.255,Z 196.746,A -85,B 0,C 180,E1 -11871.976,E2 -11871.976} C_VEL
LIN {X 0,Y 383.19,Z 196.749,A -85,B 0,C 180,E1 -11874.739,E2 -11874.739} C_VEL
LIN {X 0,Y 383.377,Z 196.731,A -85,B 0,C 180,E1 -11877.899,E2 -11877.899} C_VEL
LIN {X 0,Y 383.511,Z 196.713,A -85,B 0,C 180,E1 -11880.001,E2 -11880.001} C_VEL
LIN {X 0,Y 383.239,Z 196.745,A -85,B 0,C 180,E1 -11883.154,E2 -11883.154} C_VEL
LIN {X 0,Y 383.277,Z 196.739,A -85,B 0,C 180,E1 -11886.317,E2 -11886.317} C_VEL
LIN {X 0,Y 383.253,Z 196.742,A -85,B 0,C 180,E1 -11888.436,E2 -11888.436} C_VEL
LIN {X 0,Y 383.09,Z 196.767,A -85,B 0,C 180,E1 -11891.643,E2 -11891.643} C_VEL
LIN {X 0,Y 383.103,Z 196.762,A -85,B 0,C 180,E1 -11894.882,E2 -11894.882} C_VEL
LIN {X 0,Y 383.056,Z 196.766,A -85,B 0,C 180,E1 -11898.174,E2 -11898.174} C_VEL
LIN {X 0,Y 382.993,Z 196.779,A -85,B 0,C 180,E1 -11901.531,E2 -11901.531} C_VEL
LIN {X 0,Y 383.046,Z 196.771,A -85,B 0,C 180,E1 -11904.961,E2 -11904.961} C_VEL
LIN {X 0,Y 383.024,Z 196.77,A -85,B 0,C 180,E1 -11908.271,E2 -11908.271} C_VEL
LIN {X 0,Y 383.003,Z 196.773,A -85,B 0,C 180,E1 -11912.151,E2 -11912.151} C_VEL
LIN {X 0,Y 383.013,Z 196.773,A -85,B 0,C 180,E1 -11914.669,E2 -11914.669} C_VEL
LIN {X 0,Y 382.994,Z 196.774,A -85,B 0,C 180,E1 -11917.905,E2 -11917.905} C_VEL
LIN {X 0,Y 382.98,Z 196.779,A -85,B 0,C 180,E1 -11921.349,E2 -11921.349} C_VEL
LIN {X 0,Y 382.992,Z 196.775,A -85,B 0,C 180,E1 -11924.304,E2 -11924.304} C_VEL
LIN {X 0,Y 383.007,Z 196.776,A -85,B 0,C 180,E1 -11927.241,E2 -11927.241} C_VEL
LIN {X 0,Y 383.011,Z 196.774,A -85,B 0,C 180,E1 -11930.415,E2 -11930.415} C_VEL
LIN {X 0,Y 383.022,Z 196.771,A -85,B 0,C 180,E1 -11934.046,E2 -11934.046} C_VEL
LIN {X 0,Y 382.985,Z 196.78,A -85,B 0,C 180,E1 -11937.579,E2 -11937.579} C_VEL
LIN {X 0,Y 383.056,Z 196.972,A -85,B 0,C 180,E1 -11939.271,E2 -11939.271} C_VEL
LIN {X 0,Y 386.847,Z 213.351,A -85,B 0,C 180,E1 -11942.367,E2 -11942.367} C_VEL
LIN {X 0,Y 388.141,Z 220.583,A -85,B 0,C 180,E1 -11943.666,E2 -11943.666} C_VEL
LIN {X 0,Y 386.426,Z 240.788,A -85,B 0,C 180,E1 -11946.983,E2 -11946.983} C_VEL
LIN {X 0,Y 384.917,Z 261.829,A -85,B 0,C 180,E1 -11950.398,E2 -11950.398} C_VEL
LIN {X 0,Y 385.226,Z 266.193,A -85,B 0,C 180,E1 -11950.553,E2 -11950.553} C_VEL
LIN {X 0,Y 387.667,Z 290.477,A -85,B 0,C 180,E1 -11951.158,E2 -11951.158} C_VEL
LIN {X 0,Y 386.524,Z 368.611,A -85,B 0,C 180,E1 -11952.781,E2 -11952.781} C_VEL
LIN {X 0,Y 385.972,Z 381.943,A -85,B 0,C 180,E1 -11953.267,E2 -11953.267} C_VEL
LIN {X 0,Y 385.301,Z 394.047,A -85,B 0,C 180,E1 -11953.918,E2 -11953.918} C_VEL
LIN {X 0,Y 384.62,Z 405.781,A -85,B 0,C 180,E1 -11954.772,E2 -11954.772} C_VEL
LIN {X 0,Y 383.862,Z 417.1,A -85,B 0,C 180,E1 -11955.827,E2 -11955.827} C_VEL
LIN {X 0,Y 383.345,Z 427.246,A -85,B 0,C 180,E1 -11957.023,E2 -11957.023} C_VEL
LIN {X 0,Y 382.682,Z 436.35,A -85,B 0,C 180,E1 -11958.346,E2 -11958.346} C_VEL
LIN {X 0,Y 382.251,Z 443.84,A -85,B 0,C 180,E1 -11959.674,E2 -11959.674} C_VEL
LIN {X 0,Y 382.008,Z 451.158,A -85,B 0,C 180,E1 -11961.271,E2 -11961.271} C_VEL
LIN {X 0,Y 381.94,Z 456.063,A -85,B 0,C 180,E1 -11962.6,E2 -11962.6} C_VEL
LIN {X 0,Y 381.949,Z 460.742,A -85,B 0,C 180,E1 -11964.192,E2 -11964.192} C_VEL
LIN {X 0,Y 381.889,Z 464.211,A -85,B 0,C 180,E1 -11965.779,E2 -11965.779} C_VEL
LIN {X 0,Y 382.036,Z 465.915,A -85,B 0,C 180,E1 -11966.837,E2 -11966.837} C_VEL
LIN {X 0,Y 382.089,Z 467.172,A -85,B 0,C 180,E1 -11967.893,E2 -11967.893} C_VEL
LIN {X 0,Y 381.998,Z 467.977,A -85,B 0,C 180,E1 -11968.947,E2 -11968.947} C_VEL
LIN {X 0,Y 381.983,Z 468.312,A -85,B 0,C 180,E1 -11970.001,E2 -11970.001} C_VEL
LIN {X 0,Y 381.999,Z 468.228,A -85,B 0,C 180,E1 -11971.055,E2 -11971.055} C_VEL
LIN {X 0,Y 382.035,Z 467.73,A -85,B 0,C 180,E1 -11972.109,E2 -11972.109} C_VEL
LIN {X 0,Y 382,Z 466.757,A -85,B 0,C 180,E1 -11973.165,E2 -11973.165} C_VEL
LIN {X 0,Y 381.846,Z 465.333,A -85,B 0,C 180,E1 -11974.223,E2 -11974.223} C_VEL
LIN {X 0,Y 381.82,Z 462.017,A -85,B 0,C 180,E1 -11975.972,E2 -11975.972} C_VEL
LIN {X 0,Y 381.937,Z 458.332,A -85,B 0,C 180,E1 -11977.401,E2 -11977.401} C_VEL
LIN {X 0,Y 382.045,Z 452.12,A -85,B 0,C 180,E1 -11979.263,E2 -11979.263} C_VEL
LIN {X 0,Y 382.461,Z 445.28,A -85,B 0,C 180,E1 -11980.857,E2 -11980.857} C_VEL
LIN {X 0,Y 383.104,Z 436.794,A -85,B 0,C 180,E1 -11982.449,E2 -11982.449} C_VEL
LIN {X 0,Y 383.952,Z 427.43,A -85,B 0,C 180,E1 -11983.861,E2 -11983.861} C_VEL
LIN {X 0,Y 384.891,Z 416.188,A -85,B 0,C 180,E1 -11985.218,E2 -11985.218} C_VEL
LIN {X 0,Y 385.954,Z 405.271,A -85,B 0,C 180,E1 -11986.259,E2 -11986.259} C_VEL
LIN {X 0,Y 386.997,Z 393.103,A -85,B 0,C 180,E1 -11987.164,E2 -11987.164} C_VEL
LIN {X 0,Y 387.81,Z 381.723,A -85,B 0,C 180,E1 -11987.808,E2 -11987.808} C_VEL
LIN {X 0,Y 388.558,Z 368.861,A -85,B 0,C 180,E1 -11988.317,E2 -11988.317} C_VEL
LIN {X 0,Y 389.01,Z 348.16,A -85,B 0,C 180,E1 -11988.807,E2 -11988.807} C_VEL
LIN {X 0,Y 390.236,Z 290.028,A -85,B 0,C 180,E1 -11990.072,E2 -11990.072} C_VEL
LIN {X 0,Y 387.887,Z 269.093,A -85,B 0,C 180,E1 -11990.738,E2 -11990.738} C_VEL
LIN {X 0,Y 386.45,Z 259.713,A -85,B 0,C 180,E1 -11991.085,E2 -11991.085} C_VEL
LIN {X 0,Y 388.659,Z 233.249,A -85,B 0,C 180,E1 -11995.292,E2 -11995.292} C_VEL
LIN {X 0,Y 389.615,Z 222.814,A -85,B 0,C 180,E1 -11996.997,E2 -11996.997} C_VEL
LIN {X 0,Y 387.434,Z 212.361,A -85,B 0,C 180,E1 -11999.016,E2 -11999.016} C_VEL
LIN {X 0,Y 384.206,Z 200.94,A -85,B 0,C 180,E1 -12001.421,E2 -12001.421} C_VEL
LIN {X 0,Y 383.012,Z 196.902,A -85,B 0,C 180,E1 -12002.372,E2 -12002.372} C_VEL
LIN {X 0,Y 383.028,Z 196.775,A -85,B 0,C 180,E1 -12005.956,E2 -12005.956} C_VEL
LIN {X 0,Y 382.989,Z 196.779,A -85,B 0,C 180,E1 -12009.581,E2 -12009.581} C_VEL
LIN {X 0,Y 383.009,Z 196.776,A -85,B 0,C 180,E1 -12012.778,E2 -12012.778} C_VEL
LIN {X 0,Y 383,Z 196.775,A -85,B 0,C 180,E1 -12015.789,E2 -12015.789} C_VEL
LIN {X 0,Y 382.989,Z 196.779,A -85,B 0,C 180,E1 -12018.796,E2 -12018.796} C_VEL
LIN {X 0,Y 383.001,Z 196.774,A -85,B 0,C 180,E1 -12022.096,E2 -12022.096} C_VEL
LIN {X 0,Y 383.021,Z 196.774,A -85,B 0,C 180,E1 -12025.332,E2 -12025.332} C_VEL
LIN {X 0,Y 382.986,Z 196.778,A -85,B 0,C 180,E1 -12029.081,E2 -12029.081} C_VEL
LIN {X 0,Y 383.059,Z 196.768,A -85,B 0,C 180,E1 -12032.698,E2 -12032.698} C_VEL
LIN {X 0,Y 383.054,Z 196.768,A -85,B 0,C 180,E1 -12035.039,E2 -12035.039} C_VEL
LIN {X 0,Y 382.995,Z 196.779,A -85,B 0,C 180,E1 -12038.469,E2 -12038.469} C_VEL
LIN {X 0,Y 383.064,Z 196.769,A -85,B 0,C 180,E1 -12041.826,E2 -12041.826} C_VEL
LIN {X 0,Y 383.112,Z 196.764,A -85,B 0,C 180,E1 -12045.118,E2 -12045.118} C_VEL
LIN {X 0,Y 383.099,Z 196.767,A -85,B 0,C 180,E1 -12048.357,E2 -12048.357} C_VEL
LIN {X 0,Y 383.222,Z 196.751,A -85,B 0,C 180,E1 -12052.022,E2 -12052.022} C_VEL
LIN {X 0,Y 383.218,Z 196.926,A -85,B 0,C 180,E1 -12054.309,E2 -12054.309} C_VEL
LIN {X 0,Y 386.424,Z 208.53,A -85,B 0,C 180,E1 -12057.159,E2 -12057.159} C_VEL
LIN {X 0,Y 387.191,Z 212.686,A -85,B 0,C 180,E1 -12058.1,E2 -12058.1} C_VEL
LIN {X 0,Y 386.731,Z 224.55,A -85,B 0,C 180,E1 -12060.521,E2 -12060.521} C_VEL
LIN {X 0,Y 386.466,Z 231.561,A -85,B 0,C 180,E1 -12061.886,E2 -12061.886} C_VEL
LIN {X 0,Y 388.966,Z 242.209,A -85,B 0,C 180,E1 -12062.405,E2 -12062.405} C_VEL
LIN {X 0,Y 390.591,Z 250.412,A -85,B 0,C 180,E1 -12062.751,E2 -12062.751} C_VEL
LIN {X 0,Y 388.66,Z 316.479,A -85,B 0,C 180,E1 -12064.448,E2 -12064.448} C_VEL
LIN {X 0,Y 388.293,Z 328.758,A -85,B 0,C 180,E1 -12064.972,E2 -12064.972} C_VEL
LIN {X 0,Y 387.692,Z 340.816,A -85,B 0,C 180,E1 -12065.722,E2 -12065.722} C_VEL
LIN {X 0,Y 386.945,Z 351.838,A -85,B 0,C 180,E1 -12066.649,E2 -12066.649} C_VEL
LIN {X 0,Y 386.195,Z 361.624,A -85,B 0,C 180,E1 -12067.712,E2 -12067.712} C_VEL
LIN {X 0,Y 385.46,Z 370.364,A -85,B 0,C 180,E1 -12068.915,E2 -12068.915} C_VEL
LIN {X 0,Y 384.696,Z 377.981,A -85,B 0,C 180,E1 -12070.233,E2 -12070.233} C_VEL
LIN {X 0,Y 384.07,Z 384.32,A -85,B 0,C 180,E1 -12071.612,E2 -12071.612} C_VEL
LIN {X 0,Y 383.458,Z 389.827,A -85,B 0,C 180,E1 -12073.172,E2 -12073.172} C_VEL
LIN {X 0,Y 382.921,Z 394.235,A -85,B 0,C 180,E1 -12074.889,E2 -12074.889} C_VEL
LIN {X 0,Y 382.658,Z 396.217,A -85,B 0,C 180,E1 -12075.991,E2 -12075.991} C_VEL
LIN {X 0,Y 382.445,Z 397.646,A -85,B 0,C 180,E1 -12077.142,E2 -12077.142} C_VEL
LIN {X 0,Y 382.288,Z 398.437,A -85,B 0,C 180,E1 -12078.211,E2 -12078.211} C_VEL
LIN {X 0,Y 382.172,Z 398.663,A -85,B 0,C 180,E1 -12079.33,E2 -12079.33} C_VEL
LIN {X 0,Y 382.14,Z 398.315,A -85,B 0,C 180,E1 -12080.452,E2 -12080.452} C_VEL
LIN {X 0,Y 382.109,Z 397.398,A -85,B 0,C 180,E1 -12081.583,E2 -12081.583} C_VEL
LIN {X 0,Y 382.237,Z 395.036,A -85,B 0,C 180,E1 -12083.172,E2 -12083.172} C_VEL
LIN {X 0,Y 382.477,Z 390.776,A -85,B 0,C 180,E1 -12085,E2 -12085} C_VEL
LIN {X 0,Y 382.81,Z 384.997,A -85,B 0,C 180,E1 -12086.73,E2 -12086.73} C_VEL
LIN {X 0,Y 383.231,Z 377.84,A -85,B 0,C 180,E1 -12088.326,E2 -12088.326} C_VEL
LIN {X 0,Y 383.62,Z 370.269,A -85,B 0,C 180,E1 -12089.646,E2 -12089.646} C_VEL
LIN {X 0,Y 384.151,Z 361.935,A -85,B 0,C 180,E1 -12090.814,E2 -12090.814} C_VEL
LIN {X 0,Y 384.595,Z 352.743,A -85,B 0,C 180,E1 -12091.846,E2 -12091.846} C_VEL
LIN {X 0,Y 385.049,Z 343.158,A -85,B 0,C 180,E1 -12092.707,E2 -12092.707} C_VEL
LIN {X 0,Y 385.456,Z 332.082,A -85,B 0,C 180,E1 -12093.472,E2 -12093.472} C_VEL
LIN {X 0,Y 385.797,Z 320.202,A -85,B 0,C 180,E1 -12094.067,E2 -12094.067} C_VEL
LIN {X 0,Y 385.996,Z 308.156,A -85,B 0,C 180,E1 -12094.453,E2 -12094.453} C_VEL
LIN {X 0,Y 386.945,Z 246.721,A -85,B 0,C 180,E1 -12095.845,E2 -12095.845} C_VEL
LIN {X 0,Y 384.217,Z 229.471,A -85,B 0,C 180,E1 -12096.372,E2 -12096.372} C_VEL
LIN {X 0,Y 384.671,Z 215.519,A -85,B 0,C 180,E1 -12099.411,E2 -12099.411} C_VEL
LIN {X 0,Y 384.978,Z 208.043,A -85,B 0,C 180,E1 -12101.086,E2 -12101.086} C_VEL
LIN {X 0,Y 383.759,Z 200.415,A -85,B 0,C 180,E1 -12102.9,E2 -12102.9} C_VEL
LIN {X 0,Y 383.022,Z 196.848,A -85,B 0,C 180,E1 -12103.829,E2 -12103.829} C_VEL
LIN {X 0,Y 383.009,Z 196.777,A -85,B 0,C 180,E1 -12107.24,E2 -12107.24} C_VEL
LIN {X 0,Y 383.012,Z 196.772,A -85,B 0,C 180,E1 -12110.413,E2 -12110.413} C_VEL
LIN {X 0,Y 383.024,Z 196.773,A -85,B 0,C 180,E1 -12114.044,E2 -12114.044} C_VEL
LIN {X 0,Y 383.004,Z 196.779,A -85,B 0,C 180,E1 -12117.573,E2 -12117.573} C_VEL
LIN {X 0,Y 382.99,Z 196.775,A -85,B 0,C 180,E1 -12120.299,E2 -12120.299} C_VEL
LIN {X 0,Y 383.055,Z 196.766,A -85,B 0,C 180,E1 -12122.697,E2 -12122.697} C_VEL
LIN {X 0,Y 383.032,Z 196.77,A -85,B 0,C 180,E1 -12126.192,E2 -12126.192} C_VEL
LIN {X 0,Y 383.054,Z 196.771,A -85,B 0,C 180,E1 -12129.598,E2 -12129.598} C_VEL
LIN {X 0,Y 383.103,Z 196.763,A -85,B 0,C 180,E1 -12132.931,E2 -12132.931} C_VEL
LIN {X 0,Y 383.123,Z 196.758,A -85,B 0,C 180,E1 -12136.463,E2 -12136.463} C_VEL
LIN {X 0,Y 383.15,Z 196.755,A -85,B 0,C 180,E1 -12140.497,E2 -12140.497} C_VEL
LIN {X 0,Y 383.271,Z 196.741,A -85,B 0,C 180,E1 -12142.625,E2 -12142.625} C_VEL
LIN {X 0,Y 383.197,Z 196.751,A -85,B 0,C 180,E1 -12144.738,E2 -12144.738} C_VEL
LIN {X 0,Y 383.385,Z 196.725,A -85,B 0,C 180,E1 -12147.898,E2 -12147.898} C_VEL
LIN {X 0,Y 383.517,Z 196.709,A -85,B 0,C 180,E1 -12149.999,E2 -12149.999} C_VEL
LIN {X 0,Y 383.248,Z 196.748,A -85,B 0,C 180,E1 -12153.153,E2 -12153.153} C_VEL
LIN {X 0,Y 383.246,Z 196.742,A -85,B 0,C 180,E1 -12156.066,E2 -12156.066} C_VEL
LIN {X 0,Y 382.632,Z 196.826,A -85,B 0,C 180,E1 -12156.943,E2 -12156.943} C_VEL
LIN {X 0,Y 379.722,Z 197.183,A -85,B 0,C 180,E1 -12158.366,E2 -12158.366} C_VEL
LIN {X 0,Y 377.222,Z 197.494,A -85,B 0,C 180,E1 -12159.517,E2 -12159.517} C_VEL
LIN {X 0,Y 376.157,Z 197.627,A -85,B 0,C 180,E1 -12160.409,E2 -12160.409} C_VEL
LIN {X 0,Y 376.078,Z 197.64,A -85,B 0,C 180,E1 -12160.711,E2 -12160.711} C_VEL
LIN {X 0,Y 376.061,Z 197.638,A -85,B 0,C 180,E1 -12164.06,E2 -12164.06} C_VEL
LIN {X 0,Y 376.039,Z 197.64,A -85,B 0,C 180,E1 -12167.607,E2 -12167.607} C_VEL
LIN {X 0,Y 375.973,Z 197.654,A -85,B 0,C 180,E1 -12170.831,E2 -12170.831} C_VEL
LIN {X 0,Y 375.989,Z 197.649,A -85,B 0,C 180,E1 -12174.281,E2 -12174.281} C_VEL
LIN {X 0,Y 376.014,Z 197.65,A -85,B 0,C 180,E1 -12176.651,E2 -12176.651} C_VEL
LIN {X 0,Y 375.964,Z 197.652,A -85,B 0,C 180,E1 -12179.078,E2 -12179.078} C_VEL
LIN {X 0,Y 375.944,Z 197.656,A -85,B 0,C 180,E1 -12182.828,E2 -12182.828} C_VEL
LIN {X 0,Y 375.955,Z 197.651,A -85,B 0,C 180,E1 -12185.414,E2 -12185.414} C_VEL
LIN {X 0,Y 375.971,Z 197.653,A -85,B 0,C 180,E1 -12188.271,E2 -12188.271} C_VEL
LIN {X 0,Y 375.982,Z 197.648,A -85,B 0,C 180,E1 -12191.61,E2 -12191.61} C_VEL
LIN {X 0,Y 375.961,Z 197.65,A -85,B 0,C 180,E1 -12195.262,E2 -12195.262} C_VEL
LIN {X 0,Y 375.973,Z 197.649,A -85,B 0,C 180,E1 -12199.138,E2 -12199.138} C_VEL
LIN {X 0,Y 375.959,Z 197.653,A -85,B 0,C 180,E1 -12201.912,E2 -12201.912} C_VEL
LIN {X 0,Y 375.972,Z 197.649,A -85,B 0,C 180,E1 -12205.332,E2 -12205.332} C_VEL
LIN {X 0,Y 375.97,Z 197.653,A -85,B 0,C 180,E1 -12208.44,E2 -12208.44} C_VEL
LIN {X 0,Y 375.995,Z 197.652,A -85,B 0,C 180,E1 -12212.142,E2 -12212.142} C_VEL
LIN {X 0,Y 375.997,Z 197.647,A -85,B 0,C 180,E1 -12214.539,E2 -12214.539} C_VEL
LIN {X 0,Y 375.954,Z 197.657,A -85,B 0,C 180,E1 -12218.046,E2 -12218.046} C_VEL
LIN {X 0,Y 376.015,Z 197.645,A -85,B 0,C 180,E1 -12221.474,E2 -12221.474} C_VEL
LIN {X 0,Y 376.053,Z 197.639,A -85,B 0,C 180,E1 -12224.833,E2 -12224.833} C_VEL
LIN {X 0,Y 376.042,Z 197.643,A -85,B 0,C 180,E1 -12228.137,E2 -12228.137} C_VEL
LIN {X 0,Y 376.211,Z 197.624,A -85,B 0,C 180,E1 -12231.919,E2 -12231.919} C_VEL
LIN {X 0,Y 376.162,Z 197.625,A -85,B 0,C 180,E1 -12234.64,E2 -12234.64} C_VEL
LIN {X 0,Y 376.343,Z 197.607,A -85,B 0,C 180,E1 -12237.86,E2 -12237.86} C_VEL
LIN {X 0,Y 376.481,Z 197.588,A -85,B 0,C 180,E1 -12240.001,E2 -12240.001} C_VEL
LIN {X 0,Y 376.177,Z 197.625,A -85,B 0,C 180,E1 -12243.214,E2 -12243.214} C_VEL
LIN {X 0,Y 376.237,Z 197.616,A -85,B 0,C 180,E1 -12246.436,E2 -12246.436} C_VEL
LIN {X 0,Y 376.198,Z 197.62,A -85,B 0,C 180,E1 -12248.596,E2 -12248.596} C_VEL
LIN {X 0,Y 376.043,Z 197.642,A -85,B 0,C 180,E1 -12251.864,E2 -12251.864} C_VEL
LIN {X 0,Y 376.051,Z 197.642,A -85,B 0,C 180,E1 -12255.168,E2 -12255.168} C_VEL
LIN {X 0,Y 376.002,Z 197.645,A -85,B 0,C 180,E1 -12258.528,E2 -12258.528} C_VEL
LIN {X 0,Y 375.961,Z 197.651,A -85,B 0,C 180,E1 -12261.955,E2 -12261.955} C_VEL
LIN {X 0,Y 376.001,Z 197.65,A -85,B 0,C 180,E1 -12265.462,E2 -12265.462} C_VEL
LIN {X 0,Y 375.955,Z 197.656,A -85,B 0,C 180,E1 -12269.081,E2 -12269.081} C_VEL
LIN {X 0,Y 375.944,Z 197.655,A -85,B 0,C 180,E1 -12272.83,E2 -12272.83} C_VEL
LIN {X 0,Y 375.952,Z 197.654,A -85,B 0,C 180,E1 -12275.417,E2 -12275.417} C_VEL
LIN {X 0,Y 375.968,Z 197.649,A -85,B 0,C 180,E1 -12278.271,E2 -12278.271} C_VEL
LIN {X 0,Y 375.93,Z 197.655,A -85,B 0,C 180,E1 -12281.602,E2 -12281.602} C_VEL
LIN {X 0,Y 375.923,Z 197.658,A -85,B 0,C 180,E1 -12285.27,E2 -12285.27} C_VEL
LIN {X 0,Y 375.93,Z 197.655,A -85,B 0,C 180,E1 -12288.401,E2 -12288.401} C_VEL
LIN {X 0,Y 375.97,Z 197.649,A -85,B 0,C 180,E1 -12291.731,E2 -12291.731} C_VEL
LIN {X 0,Y 375.978,Z 197.653,A -85,B 0,C 180,E1 -12295.334,E2 -12295.334} C_VEL
LIN {X 0,Y 375.984,Z 197.794,A -85,B 0,C 180,E1 -12298.943,E2 -12298.943} C_VEL
LIN {X 0,Y 379.802,Z 214.307,A -85,B 0,C 180,E1 -12302.146,E2 -12302.146} C_VEL
LIN {X 0,Y 381.164,Z 221.347,A -85,B 0,C 180,E1 -12303.442,E2 -12303.442} C_VEL
LIN {X 0,Y 379.883,Z 236.513,A -85,B 0,C 180,E1 -12305.984,E2 -12305.984} C_VEL
LIN {X 0,Y 377.97,Z 261.532,A -85,B 0,C 180,E1 -12310.129,E2 -12310.129} C_VEL
LIN {X 0,Y 378.303,Z 266.08,A -85,B 0,C 180,E1 -12310.288,E2 -12310.288} C_VEL
LIN {X 0,Y 380.743,Z 290.96,A -85,B 0,C 180,E1 -12310.926,E2 -12310.926} C_VEL
LIN {X 0,Y 379.585,Z 367.988,A -85,B 0,C 180,E1 -12312.561,E2 -12312.561} C_VEL
LIN {X 0,Y 378.999,Z 381.333,A -85,B 0,C 180,E1 -12313.054,E2 -12313.054} C_VEL
LIN {X 0,Y 378.428,Z 392.976,A -85,B 0,C 180,E1 -12313.687,E2 -12313.687} C_VEL
LIN {X 0,Y 377.71,Z 404.007,A -85,B 0,C 180,E1 -12314.487,E2 -12314.487} C_VEL
LIN {X 0,Y 376.952,Z 415.546,A -85,B 0,C 180,E1 -12315.561,E2 -12315.561} C_VEL
LIN {X 0,Y 376.402,Z 424.368,A -85,B 0,C 180,E1 -12316.58,E2 -12316.58} C_VEL
LIN {X 0,Y 375.71,Z 433.465,A -85,B 0,C 180,E1 -12317.853,E2 -12317.853} C_VEL
LIN {X 0,Y 375.283,Z 441.354,A -85,B 0,C 180,E1 -12319.207,E2 -12319.207} C_VEL
LIN {X 0,Y 374.947,Z 449.013,A -85,B 0,C 180,E1 -12320.833,E2 -12320.833} C_VEL
LIN {X 0,Y 374.863,Z 455.122,A -85,B 0,C 180,E1 -12322.46,E2 -12322.46} C_VEL
LIN {X 0,Y 374.874,Z 459.38,A -85,B 0,C 180,E1 -12323.896,E2 -12323.896} C_VEL
LIN {X 0,Y 374.809,Z 463.41,A -85,B 0,C 180,E1 -12325.699,E2 -12325.699} C_VEL
LIN {X 0,Y 374.965,Z 465.149,A -85,B 0,C 180,E1 -12326.777,E2 -12326.777} C_VEL
LIN {X 0,Y 375.04,Z 466.432,A -85,B 0,C 180,E1 -12327.853,E2 -12327.853} C_VEL
LIN {X 0,Y 374.949,Z 467.269,A -85,B 0,C 180,E1 -12328.927,E2 -12328.927} C_VEL
LIN {X 0,Y 374.93,Z 467.633,A -85,B 0,C 180,E1 -12330.001,E2 -12330.001} C_VEL
LIN {X 0,Y 374.948,Z 467.567,A -85,B 0,C 180,E1 -12331.075,E2 -12331.075} C_VEL
LIN {X 0,Y 374.958,Z 467.086,A -85,B 0,C 180,E1 -12332.149,E2 -12332.149} C_VEL
LIN {X 0,Y 374.911,Z 466.15,A -85,B 0,C 180,E1 -12333.225,E2 -12333.225} C_VEL
LIN {X 0,Y 374.763,Z 464.747,A -85,B 0,C 180,E1 -12334.303,E2 -12334.303} C_VEL
LIN {X 0,Y 374.727,Z 461.801,A -85,B 0,C 180,E1 -12335.934,E2 -12335.934} C_VEL
LIN {X 0,Y 374.851,Z 457.827,A -85,B 0,C 180,E1 -12337.542,E2 -12337.542} C_VEL
LIN {X 0,Y 374.998,Z 451.666,A -85,B 0,C 180,E1 -12339.439,E2 -12339.439} C_VEL
LIN {X 0,Y 375.425,Z 444.871,A -85,B 0,C 180,E1 -12341.063,E2 -12341.063} C_VEL
LIN {X 0,Y 376.111,Z 436.426,A -85,B 0,C 180,E1 -12342.684,E2 -12342.684} C_VEL
LIN {X 0,Y 376.956,Z 427.849,A -85,B 0,C 180,E1 -12344.027,E2 -12344.027} C_VEL
LIN {X 0,Y 377.921,Z 417.272,A -85,B 0,C 180,E1 -12345.368,E2 -12345.368} C_VEL
LIN {X 0,Y 378.991,Z 406.819,A -85,B 0,C 180,E1 -12346.428,E2 -12346.428} C_VEL
LIN {X 0,Y 380.042,Z 395.372,A -85,B 0,C 180,E1 -12347.35,E2 -12347.35} C_VEL
LIN {X 0,Y 380.973,Z 383.575,A -85,B 0,C 180,E1 -12348.069,E2 -12348.069} C_VEL
LIN {X 0,Y 381.848,Z 370.153,A -85,B 0,C 180,E1 -12348.651,E2 -12348.651} C_VEL
LIN {X 0,Y 382.352,Z 355.185,A -85,B 0,C 180,E1 -12349.043,E2 -12349.043} C_VEL
LIN {X 0,Y 383.708,Z 290.361,A -85,B 0,C 180,E1 -12350.494,E2 -12350.494} C_VEL
LIN {X 0,Y 381.405,Z 269.817,A -85,B 0,C 180,E1 -12351.171,E2 -12351.171} C_VEL
LIN {X 0,Y 379.78,Z 259.107,A -85,B 0,C 180,E1 -12351.605,E2 -12351.605} C_VEL
LIN {X 0,Y 381.905,Z 235.661,A -85,B 0,C 180,E1 -12355.419,E2 -12355.419} C_VEL
LIN {X 0,Y 382.869,Z 224.294,A -85,B 0,C 180,E1 -12357.317,E2 -12357.317} C_VEL
LIN {X 0,Y 380.698,Z 214.107,A -85,B 0,C 180,E1 -12359.357,E2 -12359.357} C_VEL
LIN {X 0,Y 377.665,Z 203.249,A -85,B 0,C 180,E1 -12361.716,E2 -12361.716} C_VEL
LIN {X 0,Y 375.988,Z 197.772,A -85,B 0,C 180,E1 -12363.045,E2 -12363.045} C_VEL
LIN {X 0,Y 375.966,Z 197.655,A -85,B 0,C 180,E1 -12366.504,E2 -12366.504} C_VEL
LIN {X 0,Y 375.942,Z 197.657,A -85,B 0,C 180,E1 -12369.961,E2 -12369.961} C_VEL
LIN {X 0,Y 375.932,Z 197.657,A -85,B 0,C 180,E1 -12373.766,E2 -12373.766} C_VEL
LIN {X 0,Y 375.937,Z 197.657,A -85,B 0,C 180,E1 -12376.811,E2 -12376.811} C_VEL
LIN {X 0,Y 375.964,Z 197.651,A -85,B 0,C 180,E1 -12380.537,E2 -12380.537} C_VEL
LIN {X 0,Y 375.966,Z 197.652,A -85,B 0,C 180,E1 -12383.496,E2 -12383.496} C_VEL
LIN {X 0,Y 375.963,Z 197.652,A -85,B 0,C 180,E1 -12385.888,E2 -12385.888} C_VEL
LIN {X 0,Y 375.968,Z 197.653,A -85,B 0,C 180,E1 -12389.687,E2 -12389.687} C_VEL
LIN {X 0,Y 376.023,Z 197.645,A -85,B 0,C 180,E1 -12393.348,E2 -12393.348} C_VEL
LIN {X 0,Y 375.999,Z 197.647,A -85,B 0,C 180,E1 -12396.888,E2 -12396.888} C_VEL
LIN {X 0,Y 376,Z 197.651,A -85,B 0,C 180,E1 -12400.339,E2 -12400.339} C_VEL
LIN {X 0,Y 376.031,Z 197.646,A -85,B 0,C 180,E1 -12403.718,E2 -12403.718} C_VEL
LIN {X 0,Y 376.106,Z 197.636,A -85,B 0,C 180,E1 -12407.042,E2 -12407.042} C_VEL
LIN {X 0,Y 376.115,Z 197.636,A -85,B 0,C 180,E1 -12410.318,E2 -12410.318} C_VEL
LIN {X 0,Y 376.238,Z 197.792,A -85,B 0,C 180,E1 -12413.665,E2 -12413.665} C_VEL
LIN {X 0,Y 379.986,Z 211.583,A -85,B 0,C 180,E1 -12417.141,E2 -12417.141} C_VEL
LIN {X 0,Y 380.578,Z 215.617,A -85,B 0,C 180,E1 -12418.067,E2 -12418.067} C_VEL
LIN {X 0,Y 379.789,Z 231.488,A -85,B 0,C 180,E1 -12421.325,E2 -12421.325} C_VEL
LIN {X 0,Y 380.077,Z 233.187,A -85,B 0,C 180,E1 -12421.473,E2 -12421.473} C_VEL
LIN {X 0,Y 383.588,Z 248.33,A -85,B 0,C 180,E1 -12422.189,E2 -12422.189} C_VEL
LIN {X 0,Y 384.179,Z 251.909,A -85,B 0,C 180,E1 -12422.334,E2 -12422.334} C_VEL
LIN {X 0,Y 382.097,Z 316.781,A -85,B 0,C 180,E1 -12424.054,E2 -12424.054} C_VEL
LIN {X 0,Y 381.733,Z 328.494,A -85,B 0,C 180,E1 -12424.555,E2 -12424.555} C_VEL
LIN {X 0,Y 381.102,Z 340.426,A -85,B 0,C 180,E1 -12425.29,E2 -12425.29} C_VEL
LIN {X 0,Y 380.461,Z 350.287,A -85,B 0,C 180,E1 -12426.097,E2 -12426.097} C_VEL
LIN {X 0,Y 379.609,Z 360.562,A -85,B 0,C 180,E1 -12427.178,E2 -12427.178} C_VEL
LIN {X 0,Y 378.91,Z 368.742,A -85,B 0,C 180,E1 -12428.264,E2 -12428.264} C_VEL
LIN {X 0,Y 378.05,Z 376.988,A -85,B 0,C 180,E1 -12429.631,E2 -12429.631} C_VEL
LIN {X 0,Y 377.348,Z 383.528,A -85,B 0,C 180,E1 -12431.005,E2 -12431.005} C_VEL
LIN {X 0,Y 376.715,Z 388.726,A -85,B 0,C 180,E1 -12432.388,E2 -12432.388} C_VEL
LIN {X 0,Y 376.158,Z 393.469,A -85,B 0,C 180,E1 -12434.056,E2 -12434.056} C_VEL
LIN {X 0,Y 375.809,Z 395.824,A -85,B 0,C 180,E1 -12435.177,E2 -12435.177} C_VEL
LIN {X 0,Y 375.539,Z 397.554,A -85,B 0,C 180,E1 -12436.302,E2 -12436.302} C_VEL
LIN {X 0,Y 375.356,Z 398.718,A -85,B 0,C 180,E1 -12437.432,E2 -12437.432} C_VEL
LIN {X 0,Y 375.187,Z 399.283,A -85,B 0,C 180,E1 -12438.568,E2 -12438.568} C_VEL
LIN {X 0,Y 375.068,Z 398.945,A -85,B 0,C 180,E1 -12440.463,E2 -12440.463} C_VEL
LIN {X 0,Y 375.075,Z 397.485,A -85,B 0,C 180,E1 -12442.008,E2 -12442.008} C_VEL
LIN {X 0,Y 375.253,Z 394.403,A -85,B 0,C 180,E1 -12443.798,E2 -12443.798} C_VEL
LIN {X 0,Y 375.517,Z 390.01,A -85,B 0,C 180,E1 -12445.496,E2 -12445.496} C_VEL
LIN {X 0,Y 375.79,Z 384.838,A -85,B 0,C 180,E1 -12446.969,E2 -12446.969} C_VEL
LIN {X 0,Y 376.07,Z 379.27,A -85,B 0,C 180,E1 -12448.233,E2 -12448.233} C_VEL
LIN {X 0,Y 376.555,Z 371.515,A -85,B 0,C 180,E1 -12449.642,E2 -12449.642} C_VEL
LIN {X 0,Y 377.178,Z 361.979,A -85,B 0,C 180,E1 -12451.005,E2 -12451.005} C_VEL
LIN {X 0,Y 377.712,Z 351.395,A -85,B 0,C 180,E1 -12452.182,E2 -12452.182} C_VEL
LIN {X 0,Y 378.214,Z 341.165,A -85,B 0,C 180,E1 -12453.064,E2 -12453.064} C_VEL
LIN {X 0,Y 378.551,Z 330.801,A -85,B 0,C 180,E1 -12453.758,E2 -12453.758} C_VEL
LIN {X 0,Y 378.841,Z 318.701,A -85,B 0,C 180,E1 -12454.337,E2 -12454.337} C_VEL
LIN {X 0,Y 379.031,Z 305.882,A -85,B 0,C 180,E1 -12454.721,E2 -12454.721} C_VEL
LIN {X 0,Y 380.146,Z 248.19,A -85,B 0,C 180,E1 -12456.056,E2 -12456.056} C_VEL
LIN {X 0,Y 377.223,Z 229.568,A -85,B 0,C 180,E1 -12456.646,E2 -12456.646} C_VEL
LIN {X 0,Y 377.696,Z 216.282,A -85,B 0,C 180,E1 -12459.591,E2 -12459.591} C_VEL
LIN {X 0,Y 377.874,Z 207.443,A -85,B 0,C 180,E1 -12461.608,E2 -12461.608} C_VEL
LIN {X 0,Y 375.984,Z 197.753,A -85,B 0,C 180,E1 -12464.031,E2 -12464.031} C_VEL
LIN {X 0,Y 375.931,Z 197.66,A -85,B 0,C 180,E1 -12467.699,E2 -12467.699} C_VEL
LIN {X 0,Y 375.959,Z 197.65,A -85,B 0,C 180,E1 -12470.537,E2 -12470.537} C_VEL
LIN {X 0,Y 375.962,Z 197.655,A -85,B 0,C 180,E1 -12473.495,E2 -12473.495} C_VEL
LIN {X 0,Y 375.958,Z 197.654,A -85,B 0,C 180,E1 -12475.888,E2 -12475.888} C_VEL
LIN {X 0,Y 375.963,Z 197.655,A -85,B 0,C 180,E1 -12479.687,E2 -12479.687} C_VEL
LIN {X 0,Y 375.995,Z 197.647,A -85,B 0,C 180,E1 -12482.141,E2 -12482.141} C_VEL
LIN {X 0,Y 376.005,Z 197.644,A -85,B 0,C 180,E1 -12484.538,E2 -12484.538} C_VEL
LIN {X 0,Y 375.962,Z 197.651,A -85,B 0,C 180,E1 -12488.045,E2 -12488.045} C_VEL
LIN {X 0,Y 376.022,Z 197.648,A -85,B 0,C 180,E1 -12491.473,E2 -12491.473} C_VEL
LIN {X 0,Y 376.057,Z 197.64,A -85,B 0,C 180,E1 -12494.832,E2 -12494.832} C_VEL
LIN {X 0,Y 376.048,Z 197.639,A -85,B 0,C 180,E1 -12498.136,E2 -12498.136} C_VEL
LIN {X 0,Y 376.255,Z 197.614,A -85,B 0,C 180,E1 -12501.876,E2 -12501.876} C_VEL
LIN {X 0,Y 376.17,Z 197.625,A -85,B 0,C 180,E1 -12504.639,E2 -12504.639} C_VEL
LIN {X 0,Y 376.351,Z 197.602,A -85,B 0,C 180,E1 -12507.859,E2 -12507.859} C_VEL
LIN {X 0,Y 376.486,Z 197.585,A -85,B 0,C 180,E1 -12509.999,E2 -12509.999} C_VEL
LIN {X 0,Y 376.186,Z 197.626,A -85,B 0,C 180,E1 -12513.212,E2 -12513.212} C_VEL
LIN {X 0,Y 376.235,Z 197.617,A -85,B 0,C 180,E1 -12516.434,E2 -12516.434} C_VEL
LIN {X 0,Y 376.116,Z 197.631,A -85,B 0,C 180,E1 -12519.681,E2 -12519.681} C_VEL
LIN {X 0,Y 376.078,Z 197.64,A -85,B 0,C 180,E1 -12520.711,E2 -12520.711} C_VEL
LIN {X 0,Y 375.42,Z 197.727,A -85,B 0,C 180,E1 -12521.606,E2 -12521.606} C_VEL
LIN {X 0,Y 372.529,Z 198.083,A -85,B 0,C 180,E1 -12523.059,E2 -12523.059} C_VEL
LIN {X 0,Y 370.087,Z 198.383,A -85,B 0,C 180,E1 -12524.235,E2 -12524.235} C_VEL
LIN {X 0,Y 369.062,Z 198.513,A -85,B 0,C 180,E1 -12525.145,E2 -12525.145} C_VEL
LIN {X 0,Y 368.993,Z 198.519,A -85,B 0,C 180,E1 -12525.453,E2 -12525.453} C_VEL
LIN {X 0,Y 368.978,Z 198.525,A -85,B 0,C 180,E1 -12528.892,E2 -12528.892} C_VEL
LIN {X 0,Y 368.927,Z 198.529,A -85,B 0,C 180,E1 -12532.394,E2 -12532.394} C_VEL
LIN {X 0,Y 368.994,Z 198.518,A -85,B 0,C 180,E1 -12535.979,E2 -12535.979} C_VEL
LIN {X 0,Y 368.955,Z 198.527,A -85,B 0,C 180,E1 -12538.811,E2 -12538.811} C_VEL
LIN {X 0,Y 368.892,Z 198.533,A -85,B 0,C 180,E1 -12542.237,E2 -12542.237} C_VEL
LIN {X 0,Y 368.929,Z 198.528,A -85,B 0,C 180,E1 -12545.002,E2 -12545.002} C_VEL
LIN {X 0,Y 368.901,Z 198.531,A -85,B 0,C 180,E1 -12548.952,E2 -12548.952} C_VEL
LIN {X 0,Y 368.944,Z 198.527,A -85,B 0,C 180,E1 -12552.021,E2 -12552.021} C_VEL
LIN {X 0,Y 368.916,Z 198.528,A -85,B 0,C 180,E1 -12555.182,E2 -12555.182} C_VEL
LIN {X 0,Y 368.902,Z 198.534,A -85,B 0,C 180,E1 -12558.181,E2 -12558.181} C_VEL
LIN {X 0,Y 368.904,Z 198.529,A -85,B 0,C 180,E1 -12561.359,E2 -12561.359} C_VEL
LIN {X 0,Y 368.928,Z 198.526,A -85,B 0,C 180,E1 -12565.146,E2 -12565.146} C_VEL
LIN {X 0,Y 368.921,Z 198.527,A -85,B 0,C 180,E1 -12569.046,E2 -12569.046} C_VEL
LIN {X 0,Y 368.98,Z 198.521,A -85,B 0,C 180,E1 -12571.565,E2 -12571.565} C_VEL
LIN {X 0,Y 368.949,Z 198.524,A -85,B 0,C 180,E1 -12575.225,E2 -12575.225} C_VEL
LIN {X 0,Y 368.929,Z 198.526,A -85,B 0,C 180,E1 -12578.973,E2 -12578.973} C_VEL
LIN {X 0,Y 368.983,Z 198.523,A -85,B 0,C 180,E1 -12582.257,E2 -12582.257} C_VEL
LIN {X 0,Y 369.028,Z 198.517,A -85,B 0,C 180,E1 -12586.228,E2 -12586.228} C_VEL
LIN {X 0,Y 369.059,Z 198.513,A -85,B 0,C 180,E1 -12590.132,E2 -12590.132} C_VEL
LIN {X 0,Y 369.193,Z 198.496,A -85,B 0,C 180,E1 -12593.442,E2 -12593.442} C_VEL
LIN {X 0,Y 369.308,Z 198.484,A -85,B 0,C 180,E1 -12597.819,E2 -12597.819} C_VEL
LIN {X 0,Y 369.45,Z 198.464,A -85,B 0,C 180,E1 -12600.001,E2 -12600.001} C_VEL
LIN {X 0,Y 369.309,Z 198.48,A -85,B 0,C 180,E1 -12602.182,E2 -12602.182} C_VEL
LIN {X 0,Y 369.199,Z 198.492,A -85,B 0,C 180,E1 -12606.559,E2 -12606.559} C_VEL
LIN {X 0,Y 369.13,Z 198.501,A -85,B 0,C 180,E1 -12608.762,E2 -12608.762} C_VEL
LIN {X 0,Y 368.998,Z 198.518,A -85,B 0,C 180,E1 -12612.094,E2 -12612.094} C_VEL
LIN {X 0,Y 368.991,Z 198.525,A -85,B 0,C 180,E1 -12615.466,E2 -12615.466} C_VEL
LIN {X 0,Y 368.951,Z 198.525,A -85,B 0,C 180,E1 -12618.895,E2 -12618.895} C_VEL
LIN {X 0,Y 368.929,Z 198.526,A -85,B 0,C 180,E1 -12622.396,E2 -12622.396} C_VEL
LIN {X 0,Y 368.994,Z 198.518,A -85,B 0,C 180,E1 -12625.981,E2 -12625.981} C_VEL
LIN {X 0,Y 368.909,Z 198.53,A -85,B 0,C 180,E1 -12629.691,E2 -12629.691} C_VEL
LIN {X 0,Y 368.892,Z 198.536,A -85,B 0,C 180,E1 -12633.044,E2 -12633.044} C_VEL
LIN {X 0,Y 368.912,Z 198.528,A -85,B 0,C 180,E1 -12636.198,E2 -12636.198} C_VEL
LIN {X 0,Y 368.898,Z 198.535,A -85,B 0,C 180,E1 -12638.954,E2 -12638.954} C_VEL
LIN {X 0,Y 368.877,Z 198.532,A -85,B 0,C 180,E1 -12642.01,E2 -12642.01} C_VEL
LIN {X 0,Y 368.876,Z 198.537,A -85,B 0,C 180,E1 -12645.177,E2 -12645.177} C_VEL
LIN {X 0,Y 368.878,Z 198.533,A -85,B 0,C 180,E1 -12648.179,E2 -12648.179} C_VEL
LIN {X 0,Y 368.904,Z 198.531,A -85,B 0,C 180,E1 -12651.361,E2 -12651.361} C_VEL
LIN {X 0,Y 368.935,Z 198.531,A -85,B 0,C 180,E1 -12655.148,E2 -12655.148} C_VEL
LIN {X 0,Y 368.955,Z 198.728,A -85,B 0,C 180,E1 -12658.672,E2 -12658.672} C_VEL
LIN {X 0,Y 373.062,Z 216.576,A -85,B 0,C 180,E1 -12662.177,E2 -12662.177} C_VEL
LIN {X 0,Y 374.16,Z 222.065,A -85,B 0,C 180,E1 -12663.206,E2 -12663.206} C_VEL
LIN {X 0,Y 373.617,Z 230.542,A -85,B 0,C 180,E1 -12664.666,E2 -12664.666} C_VEL
LIN {X 0,Y 371.412,Z 255.678,A -85,B 0,C 180,E1 -12668.93,E2 -12668.93} C_VEL
LIN {X 0,Y 371.029,Z 261.685,A -85,B 0,C 180,E1 -12669.904,E2 -12669.904} C_VEL
LIN {X 0,Y 373.84,Z 292.065,A -85,B 0,C 180,E1 -12670.708,E2 -12670.708} C_VEL
LIN {X 0,Y 372.615,Z 367.89,A -85,B 0,C 180,E1 -12672.366,E2 -12672.366} C_VEL
LIN {X 0,Y 372.004,Z 381.06,A -85,B 0,C 180,E1 -12672.867,E2 -12672.867} C_VEL
LIN {X 0,Y 371.424,Z 392.619,A -85,B 0,C 180,E1 -12673.512,E2 -12673.512} C_VEL
LIN {X 0,Y 370.599,Z 405.199,A -85,B 0,C 180,E1 -12674.464,E2 -12674.464} C_VEL
LIN {X 0,Y 369.805,Z 416.401,A -85,B 0,C 180,E1 -12675.557,E2 -12675.557} C_VEL
LIN {X 0,Y 369.305,Z 425.008,A -85,B 0,C 180,E1 -12676.598,E2 -12676.598} C_VEL
LIN {X 0,Y 368.6,Z 433.832,A -85,B 0,C 180,E1 -12677.894,E2 -12677.894} C_VEL
LIN {X 0,Y 368.176,Z 441.554,A -85,B 0,C 180,E1 -12679.275,E2 -12679.275} C_VEL
LIN {X 0,Y 367.852,Z 449.074,A -85,B 0,C 180,E1 -12680.932,E2 -12680.932} C_VEL
LIN {X 0,Y 367.811,Z 454.131,A -85,B 0,C 180,E1 -12682.314,E2 -12682.314} C_VEL
LIN {X 0,Y 367.81,Z 458.761,A -85,B 0,C 180,E1 -12683.891,E2 -12683.891} C_VEL
LIN {X 0,Y 367.735,Z 462.563,A -85,B 0,C 180,E1 -12685.616,E2 -12685.616} C_VEL
LIN {X 0,Y 367.895,Z 464.359,A -85,B 0,C 180,E1 -12686.715,E2 -12686.715} C_VEL
LIN {X 0,Y 367.991,Z 465.67,A -85,B 0,C 180,E1 -12687.812,E2 -12687.812} C_VEL
LIN {X 0,Y 367.901,Z 466.532,A -85,B 0,C 180,E1 -12688.906,E2 -12688.906} C_VEL
LIN {X 0,Y 367.879,Z 466.947,A -85,B 0,C 180,E1 -12690.001,E2 -12690.001} C_VEL
LIN {X 0,Y 367.898,Z 466.906,A -85,B 0,C 180,E1 -12691.095,E2 -12691.095} C_VEL
LIN {X 0,Y 367.883,Z 466.442,A -85,B 0,C 180,E1 -12692.19,E2 -12692.19} C_VEL
LIN {X 0,Y 367.826,Z 465.548,A -85,B 0,C 180,E1 -12693.287,E2 -12693.287} C_VEL
LIN {X 0,Y 367.682,Z 464.168,A -85,B 0,C 180,E1 -12694.386,E2 -12694.386} C_VEL
LIN {X 0,Y 367.71,Z 460.634,A -85,B 0,C 180,E1 -12696.344,E2 -12696.344} C_VEL
LIN {X 0,Y 367.764,Z 455.755,A -85,B 0,C 180,E1 -12698.241,E2 -12698.241} C_VEL
LIN {X 0,Y 368.047,Z 449.114,A -85,B 0,C 180,E1 -12700.174,E2 -12700.174} C_VEL
LIN {X 0,Y 368.677,Z 441.937,A -85,B 0,C 180,E1 -12701.826,E2 -12701.826} C_VEL
LIN {X 0,Y 369.514,Z 432.972,A -85,B 0,C 180,E1 -12703.47,E2 -12703.47} C_VEL
LIN {X 0,Y 370.521,Z 422.74,A -85,B 0,C 180,E1 -12704.978,E2 -12704.978} C_VEL
LIN {X 0,Y 371.577,Z 412.311,A -85,B 0,C 180,E1 -12706.2,E2 -12706.2} C_VEL
LIN {X 0,Y 372.848,Z 400.769,A -85,B 0,C 180,E1 -12707.271,E2 -12707.271} C_VEL
LIN {X 0,Y 373.877,Z 388.668,A -85,B 0,C 180,E1 -12708.14,E2 -12708.14} C_VEL
LIN {X 0,Y 374.93,Z 375.396,A -85,B 0,C 180,E1 -12708.831,E2 -12708.831} C_VEL
LIN {X 0,Y 375.577,Z 363.352,A -85,B 0,C 180,E1 -12709.258,E2 -12709.258} C_VEL
LIN {X 0,Y 377.264,Z 291.042,A -85,B 0,C 180,E1 -12710.932,E2 -12710.932} C_VEL
LIN {X 0,Y 375.163,Z 271.902,A -85,B 0,C 180,E1 -12711.584,E2 -12711.584} C_VEL
LIN {X 0,Y 373.132,Z 258.696,A -85,B 0,C 180,E1 -12712.13,E2 -12712.13} C_VEL
LIN {X 0,Y 375.429,Z 235.226,A -85,B 0,C 180,E1 -12716.03,E2 -12716.03} C_VEL
LIN {X 0,Y 376.277,Z 226.452,A -85,B 0,C 180,E1 -12717.534,E2 -12717.534} C_VEL
LIN {X 0,Y 373.98,Z 215.841,A -85,B 0,C 180,E1 -12719.715,E2 -12719.715} C_VEL
LIN {X 0,Y 370.685,Z 204.256,A -85,B 0,C 180,E1 -12722.338,E2 -12722.338} C_VEL
LIN {X 0,Y 368.948,Z 198.631,A -85,B 0,C 180,E1 -12723.779,E2 -12723.779} C_VEL
LIN {X 0,Y 368.901,Z 198.535,A -85,B 0,C 180,E1 -12727.564,E2 -12727.564} C_VEL
LIN {X 0,Y 368.886,Z 198.537,A -85,B 0,C 180,E1 -12730.374,E2 -12730.374} C_VEL
LIN {X 0,Y 368.885,Z 198.536,A -85,B 0,C 180,E1 -12733.616,E2 -12733.616} C_VEL
LIN {X 0,Y 368.889,Z 198.534,A -85,B 0,C 180,E1 -12736.696,E2 -12736.696} C_VEL
LIN {X 0,Y 368.913,Z 198.529,A -85,B 0,C 180,E1 -12739.643,E2 -12739.643} C_VEL
LIN {X 0,Y 368.904,Z 198.535,A -85,B 0,C 180,E1 -12743.144,E2 -12743.144} C_VEL
LIN {X 0,Y 368.9,Z 198.53,A -85,B 0,C 180,E1 -12746.462,E2 -12746.462} C_VEL
LIN {X 0,Y 368.932,Z 198.528,A -85,B 0,C 180,E1 -12749.046,E2 -12749.046} C_VEL
LIN {X 0,Y 368.966,Z 198.523,A -85,B 0,C 180,E1 -12752.796,E2 -12752.796} C_VEL
LIN {X 0,Y 368.948,Z 198.528,A -85,B 0,C 180,E1 -12756.113,E2 -12756.113} C_VEL
LIN {X 0,Y 368.939,Z 198.529,A -85,B 0,C 180,E1 -12759.947,E2 -12759.947} C_VEL
LIN {X 0,Y 368.978,Z 198.524,A -85,B 0,C 180,E1 -12763.398,E2 -12763.398} C_VEL
LIN {X 0,Y 369.06,Z 198.515,A -85,B 0,C 180,E1 -12766.79,E2 -12766.79} C_VEL
LIN {X 0,Y 369.065,Z 198.514,A -85,B 0,C 180,E1 -12770.131,E2 -12770.131} C_VEL
LIN {X 0,Y 369.155,Z 198.696,A -85,B 0,C 180,E1 -12772.96,E2 -12772.96} C_VEL
LIN {X 0,Y 371.968,Z 208.911,A -85,B 0,C 180,E1 -12775.665,E2 -12775.665} C_VEL
LIN {X 0,Y 373.823,Z 216.167,A -85,B 0,C 180,E1 -12777.476,E2 -12777.476} C_VEL
LIN {X 0,Y 373.824,Z 221.688,A -85,B 0,C 180,E1 -12778.679,E2 -12778.679} C_VEL
LIN {X 0,Y 373.174,Z 232.298,A -85,B 0,C 180,E1 -12780.864,E2 -12780.864} C_VEL
LIN {X 0,Y 377.083,Z 248.92,A -85,B 0,C 180,E1 -12781.718,E2 -12781.718} C_VEL
LIN {X 0,Y 377.742,Z 253.676,A -85,B 0,C 180,E1 -12781.907,E2 -12781.907} C_VEL
LIN {X 0,Y 375.578,Z 317.808,A -85,B 0,C 180,E1 -12783.654,E2 -12783.654} C_VEL
LIN {X 0,Y 375.172,Z 329.294,A -85,B 0,C 180,E1 -12784.162,E2 -12784.162} C_VEL
LIN {X 0,Y 374.476,Z 341.447,A -85,B 0,C 180,E1 -12784.934,E2 -12784.934} C_VEL
LIN {X 0,Y 373.759,Z 351.625,A -85,B 0,C 180,E1 -12785.8,E2 -12785.8} C_VEL
LIN {X 0,Y 372.851,Z 361.741,A -85,B 0,C 180,E1 -12786.901,E2 -12786.901} C_VEL
LIN {X 0,Y 372.004,Z 370.718,A -85,B 0,C 180,E1 -12788.145,E2 -12788.145} C_VEL
LIN {X 0,Y 371.196,Z 378.139,A -85,B 0,C 180,E1 -12789.423,E2 -12789.423} C_VEL
LIN {X 0,Y 370.382,Z 385.044,A -85,B 0,C 180,E1 -12790.938,E2 -12790.938} C_VEL
LIN {X 0,Y 369.625,Z 390.946,A -85,B 0,C 180,E1 -12792.63,E2 -12792.63} C_VEL
LIN {X 0,Y 369.021,Z 395.263,A -85,B 0,C 180,E1 -12794.334,E2 -12794.334} C_VEL
LIN {X 0,Y 368.707,Z 397.325,A -85,B 0,C 180,E1 -12795.477,E2 -12795.477} C_VEL
LIN {X 0,Y 368.452,Z 398.817,A -85,B 0,C 180,E1 -12796.625,E2 -12796.625} C_VEL
LIN {X 0,Y 368.235,Z 399.715,A -85,B 0,C 180,E1 -12797.78,E2 -12797.78} C_VEL
LIN {X 0,Y 368.081,Z 400.031,A -85,B 0,C 180,E1 -12798.94,E2 -12798.94} C_VEL
LIN {X 0,Y 368.001,Z 399.466,A -85,B 0,C 180,E1 -12800.643,E2 -12800.643} C_VEL
LIN {X 0,Y 368.022,Z 397.47,A -85,B 0,C 180,E1 -12802.453,E2 -12802.453} C_VEL
LIN {X 0,Y 368.245,Z 394.096,A -85,B 0,C 180,E1 -12804.225,E2 -12804.225} C_VEL
LIN {X 0,Y 368.537,Z 389.065,A -85,B 0,C 180,E1 -12806.015,E2 -12806.015} C_VEL
LIN {X 0,Y 368.834,Z 383.425,A -85,B 0,C 180,E1 -12807.52,E2 -12807.52} C_VEL
LIN {X 0,Y 369.235,Z 376.931,A -85,B 0,C 180,E1 -12808.888,E2 -12808.888} C_VEL
LIN {X 0,Y 369.741,Z 368.899,A -85,B 0,C 180,E1 -12810.245,E2 -12810.245} C_VEL
LIN {X 0,Y 370.241,Z 360.249,A -85,B 0,C 180,E1 -12811.414,E2 -12811.414} C_VEL
LIN {X 0,Y 370.824,Z 349.831,A -85,B 0,C 180,E1 -12812.532,E2 -12812.532} C_VEL
LIN {X 0,Y 371.303,Z 339.309,A -85,B 0,C 180,E1 -12813.412,E2 -12813.412} C_VEL
LIN {X 0,Y 371.789,Z 327.459,A -85,B 0,C 180,E1 -12814.146,E2 -12814.146} C_VEL
LIN {X 0,Y 371.957,Z 315.202,A -85,B 0,C 180,E1 -12814.673,E2 -12814.673} C_VEL
LIN {X 0,Y 372.662,Z 275.09,A -85,B 0,C 180,E1 -12815.658,E2 -12815.658} C_VEL
LIN {X 0,Y 373.175,Z 248.512,A -85,B 0,C 180,E1 -12816.301,E2 -12816.301} C_VEL
LIN {X 0,Y 370.291,Z 230.052,A -85,B 0,C 180,E1 -12816.887,E2 -12816.887} C_VEL
LIN {X 0,Y 370.51,Z 223.082,A -85,B 0,C 180,E1 -12818.404,E2 -12818.404} C_VEL
LIN {X 0,Y 370.992,Z 209.425,A -85,B 0,C 180,E1 -12821.531,E2 -12821.531} C_VEL
LIN {X 0,Y 368.947,Z 198.752,A -85,B 0,C 180,E1 -12824.197,E2 -12824.197} C_VEL
LIN {X 0,Y 368.884,Z 198.536,A -85,B 0,C 180,E1 -12826.695,E2 -12826.695} C_VEL
LIN {X 0,Y 368.91,Z 198.534,A -85,B 0,C 180,E1 -12829.642,E2 -12829.642} C_VEL
LIN {X 0,Y 368.899,Z 198.531,A -85,B 0,C 180,E1 -12833.144,E2 -12833.144} C_VEL
LIN {X 0,Y 368.897,Z 198.53,A -85,B 0,C 180,E1 -12836.461,E2 -12836.461} C_VEL
LIN {X 0,Y 368.928,Z 198.528,A -85,B 0,C 180,E1 -12839.046,E2 -12839.046} C_VEL
LIN {X 0,Y 368.978,Z 198.526,A -85,B 0,C 180,E1 -12841.563,E2 -12841.563} C_VEL
LIN {X 0,Y 368.998,Z 198.519,A -85,B 0,C 180,E1 -12844.019,E2 -12844.019} C_VEL
LIN {X 0,Y 368.931,Z 198.53,A -85,B 0,C 180,E1 -12847.604,E2 -12847.604} C_VEL
LIN {X 0,Y 368.981,Z 198.523,A -85,B 0,C 180,E1 -12851.107,E2 -12851.107} C_VEL
LIN {X 0,Y 368.996,Z 198.518,A -85,B 0,C 180,E1 -12854.534,E2 -12854.534} C_VEL
LIN {X 0,Y 369.003,Z 198.518,A -85,B 0,C 180,E1 -12857.906,E2 -12857.906} C_VEL
LIN {X 0,Y 369.227,Z 198.49,A -85,B 0,C 180,E1 -12861.8,E2 -12861.8} C_VEL
LIN {X 0,Y 369.143,Z 198.5,A -85,B 0,C 180,E1 -12864.537,E2 -12864.537} C_VEL
LIN {X 0,Y 369.316,Z 198.478,A -85,B 0,C 180,E1 -12867.818,E2 -12867.818} C_VEL
LIN {X 0,Y 369.456,Z 198.46,A -85,B 0,C 180,E1 -12869.999,E2 -12869.999} C_VEL
LIN {X 0,Y 369.316,Z 198.478,A -85,B 0,C 180,E1 -12872.18,E2 -12872.18} C_VEL
LIN {X 0,Y 369.195,Z 198.495,A -85,B 0,C 180,E1 -12876.558,E2 -12876.558} C_VEL
